# B&R Automation Studio project NAEUL004C00R13L518F00 (part 22)

#### Act_OptP0938FBCtrl1.st
```iecst
ACTION Act_OptP0938FBCtrl1:

	//Motor
	fbJogSlowToFastDlyTm.PT	:= T#2s;
	fbJogSlowToFastDlyTm;
	fbLmtRstTm;

	IF EDGENEG(bMagAWSelfTest) THEN
		eMag1AWEngageAct	:= PneuActIdle;
		eMagAWOpen1Act	:= MagAWActIdle;
	END_IF

	IF bMagAWSelfTest = FALSE THEN

		usiMagAWSelfTestStep := 0;
		//Interruption
		IF tyP0938MagAW.tyMagAW1.tyBtnMtrGearEngage.bRtCompl = TRUE AND (EDGENEG(p_tyDI.bMagPresentSen1) OR EDGEPOS(p_eMag1AWEngageStatus = Error)) THEN
			tyP0938MagAW.tyMotionStd1.tyBtnStop.bRtCompl	:= TRUE;
		END_IF

		IF EDGEPOS((p_udiMagAWOpen1AxisErrID = 21570 OR p_udiMagAWOpen1AxisErrID = 21571) AND tyP0938MagAW.tyMotionStd1.tyBtnJogOpen.bValue = FALSE AND tyP0938MagAW.tyMotionStd1.tyBtnJogClose.bValue = FALSE) THEN
			fbLmtRstTm.IN	:= TRUE;
		END_IF

		IF fbLmtRstTm.Q = TRUE THEN
			tyP0938MagAW.tyMotionStd1.tyBtnRst.bRtCompl		:= TRUE;
		END_IF

		IF (tyP0938MagAW.tyMotionStd1.tyBtnJogOpen.bValue = FALSE AND tyP0938MagAW.tyMotionStd1.tyBtnJogClose.bValue = FALSE) AND (p_bMagAWOpen1Jogging = TRUE) THEN
			bJogStopMagAW1	:= TRUE;
		END_IF

		IF tyP0938MagAW.tyMotionStd1.tyBtnStop.bRtCompl = TRUE THEN

			IF tyP0938MagAW.tyMagAW1.tyBtnMtrGearEngage.bRtCompl = TRUE THEN
				eMagAWOpen1Act		:= MagAWActEngageStop;
				eMag1AWEngageAct	:= PneuActIdle;
			ELSE
				eMagAWOpen1Act		:= MagAWActStop;
			END_IF

			IF (p_eMagAWOpen1Stat = MagAWActStop AND p_eMagAWOpen1Status = Done) OR (p_eMagAWOpen1Stat = MagAWActEngageStop AND p_eMagAWOpen1Status = Done) THEN
				eMagAWOpen1Act	:= MagAWActIdle;

				tyP0938MagAW.tyMotionStd1.tyBtnStop.bRtCompl		:= FALSE;
				tyP0938MagAW.tyMotionStd1.tyBtnJogOpen.bRtCompl		:= FALSE;
				tyP0938MagAW.tyMotionStd1.tyBtnJogClose.bRtCompl	:= FALSE;
				tyP0938MagAW.tyMotionStd1.tyBtnOrigin.bRtCompl		:= FALSE;
				tyP0938MagAW.tyMotionStd1.tyBtnMovAbs.bRtCompl		:= FALSE;
				tyP0938MagAW.tyMotionStd1.tyBtnMovRel.bRtCompl		:= FALSE;
				tyP0938MagAW.tyMagAW1.tyBtnGo.bRtCompl				:= FALSE;
				tyP0938MagAW.tyMagAW1.tyBtnMtrGearEngage.bRtCompl	:= FALSE;

				tyP0938MagAW.tyMotionStd1.tyBtnStop.bValue			:= TRUE;
				tyP0938MagAW.tyMotionStd1.tyBtnJogOpen.bValue		:= FALSE;
				tyP0938MagAW.tyMotionStd1.tyBtnJogClose.bValue		:= FALSE;
				tyP0938MagAW.tyMotionStd1.tyBtnOrigin.bValue		:= FALSE;
				tyP0938MagAW.tyMotionStd1.tyBtnMovAbs.bValue		:= FALSE;
				tyP0938MagAW.tyMotionStd1.tyBtnMovRel.bValue		:= FALSE;
				tyP0938MagAW.tyMagAW1.tyBtnGo.bValue				:= FALSE;
				tyP0938MagAW.tyMagAW1.tyBtnMtrGearEngage.bValue		:= FALSE;

				tyP0938MagAW.tyMotionStd1.tyBtnStop.bRtLk			:= TRUE;
				tyP0938MagAW.tyMotionStd1.tyBtnJogOpen.bRtLk		:= FALSE;
				tyP0938MagAW.tyMotionStd1.tyBtnJogClose.bRtLk		:= FALSE;
				tyP0938MagAW.tyMotionStd1.tyBtnOrigin.bRtLk			:= FALSE;
				tyP0938MagAW.tyMotionStd1.tyBtnMovAbs.bRtLk			:= FALSE;
				tyP0938MagAW.tyMotionStd1.tyBtnMovRel.bRtLk			:= FALSE;
				tyP0938MagAW.tyMagAW1.tyBtnGo.bRtLk					:= FALSE;
				tyP0938MagAW.tyMagAW1.tyBtnMtrGearEngage.bRtLk		:= FALSE;
			END_IF

		ELSIF (tyP0938MagAW.tyMotionStd1.tyBtnJogOpen.bRtCompl = TRUE) OR (tyP0938MagAW.tyMotionStd1.tyBtnJogClose.bRtCompl = TRUE) OR (bJogStopMagAW1 = TRUE) THEN
			bJogSlow					:= FALSE;
			bJogFast					:= FALSE;
			fbJogSlowToFastDlyTm.IN		:= FALSE;

			eMagAWOpen1Act	:= MagAWActJogStop;

			IF p_eMagAWOpen1Stat = MagAWActJogStop AND p_eMagAWOpen1Status = Done THEN
				eMagAWOpen1Act	:= MagAWActIdle;

				bJogStopMagAW1	:= FALSE;

				tyP0938MagAW.tyMotionStd1.tyBtnStop.bRtCompl		:= FALSE;
				tyP0938MagAW.tyMotionStd1.tyBtnJogOpen.bRtCompl		:= FALSE;
				tyP0938MagAW.tyMotionStd1.tyBtnJogClose.bRtCompl	:= FALSE;
				tyP0938MagAW.tyMotionStd1.tyBtnOrigin.bRtCompl		:= FALSE;
				tyP0938MagAW.tyMotionStd1.tyBtnMovAbs.bRtCompl		:= FALSE;
				tyP0938MagAW.tyMotionStd1.tyBtnMovRel.bRtCompl		:= FALSE;
				tyP0938MagAW.tyMagAW1.tyBtnGo.bRtCompl				:= FALSE;

				tyP0938MagAW.tyMotionStd1.tyBtnStop.bValue			:= TRUE;
				tyP0938MagAW.tyMotionStd1.tyBtnJogOpen.bValue		:= FALSE;
				tyP0938MagAW.tyMotionStd1.tyBtnJogClose.bValue		:= FALSE;
				tyP0938MagAW.tyMotionStd1.tyBtnOrigin.bValue		:= FALSE;
				tyP0938MagAW.tyMotionStd1.tyBtnMovAbs.bValue		:= FALSE;
				tyP0938MagAW.tyMotionStd1.tyBtnMovRel.bValue		:= FALSE;
				tyP0938MagAW.tyMagAW1.tyBtnGo.bValue				:= FALSE;

				tyP0938MagAW.tyMotionStd1.tyBtnStop.bRtLk			:= TRUE;
				tyP0938MagAW.tyMotionStd1.tyBtnJogOpen.bRtLk		:= FALSE;
				tyP0938MagAW.tyMotionStd1.tyBtnJogClose.bRtLk		:= FALSE;
				tyP0938MagAW.tyMotionStd1.tyBtnOrigin.bRtLk			:= FALSE;
				tyP0938MagAW.tyMotionStd1.tyBtnMovAbs.bRtLk			:= FALSE;
				tyP0938MagAW.tyMotionStd1.tyBtnMovRel.bRtLk			:= FALSE;
				tyP0938MagAW.tyMagAW1.tyBtnGo.bRtLk					:= FALSE;
			END_IF

		ELSIF tyP0938MagAW.tyMotionStd1.tyBtnPwr.bRtCompl = TRUE THEN
			tyP0938MagAW.tyMotionStd1.tyBtnPwr.bRtLk	:= TRUE;

			IF tyP0938MagAW.tyMotionStd1.tyBtnPwr.bValue = TRUE THEN
				eMagAWOpen1Act	:= MagAWActPwrOn;

				IF p_eMagAWOpen1Stat = MagAWActPwrOn AND p_eMagAWOpen1Status = Done THEN
					eMagAWOpen1Act	:= MagAWActIdle;

					tyP0938MagAW.tyMotionStd1.tyBtnPwr.bRtCompl	:= FALSE;
					tyP0938MagAW.tyMotionStd1.tyBtnPwr.bRtLk	:= FALSE;
				END_IF
			ELSE
				eMagAWOpen1Act	:= MagAWActPwrOff;

				IF p_eMagAWOpen1Stat = MagAWActPwrOff AND p_eMagAWOpen1Status = Done THEN
					eMagAWOpen1Act	:= MagAWActIdle;

					tyP0938MagAW.tyMotionStd1.tyBtnPwr.bRtCompl	:= FALSE;
					tyP0938MagAW.tyMotionStd1.tyBtnPwr.bRtLk	:= FALSE;
				END_IF
			END_IF

		ELSIF tyP0938MagAW.tyMotionStd1.tyBtnOrigin.bRtCompl = TRUE THEN
			tyP0938MagAW.tyMotionStd1.tyBtnOrigin.bValue	:= TRUE;
			tyP0938MagAW.tyMotionStd1.tyBtnStop.bValue		:= FALSE;

			tyP0938MagAW.tyMotionStd1.tyBtnOrigin.bRtLk		:= TRUE;
			tyP0938MagAW.tyMotionStd1.tyBtnStop.bRtLk		:= FALSE;

			eMagAWOpen1Act	:= MagAWActHoming;

			IF p_eMagAWOpen1Stat = MagAWActHoming AND p_eMagAWOpen1Status = Done THEN
				eMagAWOpen1Act	:= MagAWActIdle;

				tyP0938MagAW.tyMotionStd1.tyBtnOrigin.bRtCompl	:= FALSE;
				tyP0938MagAW.tyMotionStd1.tyBtnOrigin.bValue	:= FALSE;
				tyP0938MagAW.tyMotionStd1.tyBtnStop.bValue		:= TRUE;

				tyP0938MagAW.tyMotionStd1.tyBtnOrigin.bRtLk		:= FALSE;
				tyP0938MagAW.tyMotionStd1.tyBtnStop.bRtLk		:= TRUE;
			END_IF

		ELSIF tyP0938MagAW.tyMotionStd1.tyBtnRst.bRtCompl = TRUE THEN
			tyP0938MagAW.tyMotionStd1.tyBtnRst.bValue	:= TRUE;
			tyP0938MagAW.tyMotionStd1.tyBtnRst.bRtLk	:= TRUE;

			eMagAWOpen1Act	:= MagAWActRstAxisErr;

			IF p_eMagAWOpen1Stat = MagAWActRstAxisErr AND p_eMagAWOpen1Status = Done THEN
				eMagAWOpen1Act	:= MagAWActIdle;

				tyP0938MagAW.tyMotionStd1.tyBtnRst.bRtCompl	:= FALSE;
				tyP0938MagAW.tyMotionStd1.tyBtnRst.bValue	:= FALSE;
				tyP0938MagAW.tyMotionStd1.tyBtnRst.bRtLk	:= FALSE;

				fbLmtRstTm.IN	:= FALSE;
			END_IF

		ELSIF tyP0938MagAW.tyMagAW1.tyBtnGo.bRtCompl = TRUE THEN
			tyP0938MagAW.tyMagAW1.tyBtnGo.bValue		:= TRUE;
			tyP0938MagAW.tyMotionStd1.tyBtnStop.bValue	:= FALSE;

			tyP0938MagAW.tyMagAW1.tyBtnGo.bRtLk			:= TRUE;
			tyP0938MagAW.tyMotionStd1.tyBtnStop.bRtLk	:= FALSE;

			diMnlMagAW1GoWidth	:= tyP0938MagAW.tyMagAW1.tyNumNewWidth.diValue;
			diMnlMagAW1NomSpd	:= tyP0938MagAW.tyMotionStd1.tyNumNomSpd.diValue;

			eMagAWOpen1Act	:= MagAWActGoWidth;

			IF p_eMagAWOpen1Stat = MagAWActGoWidth AND p_eMagAWOpen1Status = Done THEN
				eMagAWOpen1Act	:= MagAWActIdle;

				tyP0938MagAW.tyMagAW1.tyBtnGo.bRtCompl		:= FALSE;
				tyP0938MagAW.tyMagAW1.tyBtnGo.bValue		:= FALSE;
				tyP0938MagAW.tyMotionStd1.tyBtnStop.bValue	:= TRUE;

				tyP0938MagAW.tyMagAW1.tyBtnGo.bRtLk			:= FALSE;
				tyP0938MagAW.tyMotionStd1.tyBtnStop.bRtLk	:= TRUE;
			END_IF

		ELSIF tyP0938MagAW.tyMotionStd1.tyBtnMovAbs.bRtCompl = TRUE THEN
			tyP0938MagAW.tyMotionStd1.tyBtnMovAbs.bValue	:= TRUE;
			tyP0938MagAW.tyMotionStd1.tyBtnStop.bValue		:= FALSE;

			tyP0938MagAW.tyMotionStd1.tyBtnMovAbs.bRtLk		:= TRUE;
			tyP0938MagAW.tyMotionStd1.tyBtnStop.bRtLk		:= FALSE;

			diMnlMagAW1TargetPos	:= tyP0938MagAW.tyMotionStd1.tyNumTargetPos.diValue;
			diMnlMagAW1NomSpd		:= tyP0938MagAW.tyMotionStd1.tyNumNomSpd.diValue;

			eMagAWOpen1Act	:= MagAWActMovAbs;

			IF p_eMagAWOpen1Stat = MagAWActMovAbs AND p_eMagAWOpen1Status = Done THEN
				eMagAWOpen1Act	:= MagAWActIdle;

				tyP0938MagAW.tyMotionStd1.tyBtnMovAbs.bRtCompl	:= FALSE;
				tyP0938MagAW.tyMotionStd1.tyBtnMovAbs.bValue	:= FALSE;
				tyP0938MagAW.tyMotionStd1.tyBtnStop.bValue		:= TRUE;

				tyP0938MagAW.tyMotionStd1.tyBtnMovAbs.bRtLk		:= FALSE;
				tyP0938MagAW.tyMotionStd1.tyBtnStop.bRtLk		:= TRUE;
			END_IF

		ELSIF tyP0938MagAW.tyMotionStd1.tyBtnMovRel.bRtCompl = TRUE THEN
			tyP0938MagAW.tyMotionStd1.tyBtnMovRel.bValue	:= TRUE;
			tyP0938MagAW.tyMotionStd1.tyBtnStop.bValue		:= FALSE;

			tyP0938MagAW.tyMotionStd1.tyBtnMovRel.bRtLk		:= TRUE;
			tyP0938MagAW.tyMotionStd1.tyBtnStop.bRtLk		:= FALSE;

			diMnlMagAW1StepSize	:= tyP0938MagAW.tyMotionStd1.tyNumStepSize.diValue;
			diMnlMagAW1NomSpd	:= tyP0938MagAW.tyMotionStd1.tyNumNomSpd.diValue;

			eMagAWOpen1Act	:= MagAWActMovRel;

			IF p_eMagAWOpen1Stat = MagAWActMovRel AND p_eMagAWOpen1Status = Done THEN
				eMagAWOpen1Act	:= MagAWActIdle;

				tyP0938MagAW.tyMotionStd1.tyBtnMovRel.bRtCompl	:= FALSE;
				tyP0938MagAW.tyMotionStd1.tyBtnMovRel.bValue	:= FALSE;
				tyP0938MagAW.tyMotionStd1.tyBtnStop.bValue		:= TRUE;

				tyP0938MagAW.tyMotionStd1.tyBtnMovRel.bRtLk		:= FALSE;
				tyP0938MagAW.tyMotionStd1.tyBtnStop.bRtLk		:= TRUE;
			END_IF

		ELSIF (tyP0938MagAW.tyMotionStd1.tyBtnJogOpen.bValue = TRUE) AND (fbJogSlowToFastDlyTm.Q = FALSE) AND (bJogSlow = FALSE) THEN
			tyP0938MagAW.tyMotionStd1.tyBtnStop.bValue	:= FALSE;
			tyP0938MagAW.tyMotionStd1.tyBtnStop.bRtLk	:= FALSE;

			fbJogSlowToFastDlyTm.IN	:= TRUE;

			diMnlMagAW1JogSpd	:= tyP0938MagAW.tyMotionStd1.tyNumSlwSpd.diValue;

			eMagAWOpen1Act	:= MagAWActJogOpen;

			IF p_eMagAWOpen1Stat = MagAWActJogOpen AND p_eMagAWOpen1Status = Done THEN
				eMagAWOpen1Act				:= MagAWActIdle;
				bJogSlow				:= TRUE;
			ELSIF p_eMagAWOpen1Status = Error THEN
				fbJogSlowToFastDlyTm.IN	:= FALSE;
				bJogSlow				:= TRUE;
			END_IF

		ELSIF (tyP0938MagAW.tyMotionStd1.tyBtnJogOpen.bValue = TRUE) AND (fbJogSlowToFastDlyTm.Q = TRUE) AND (bJogFast = FALSE) THEN
			tyP0938MagAW.tyMotionStd1.tyBtnStop.bValue	:= FALSE;
			tyP0938MagAW.tyMotionStd1.tyBtnStop.bRtLk	:= FALSE;

			fbJogSlowToFastDlyTm.IN	:= TRUE;

			diMnlMagAW1JogSpd	:= tyP0938MagAW.tyMotionStd1.tyNumNomSpd.diValue;

			eMagAWOpen1Act	:= MagAWActJogOpen;

			IF p_eMagAWOpen1Stat = MagAWActJogOpen AND p_eMagAWOpen1Status = Done THEN
				eMagAWOpen1Act				:= MagAWActIdle;
				bJogFast				:= TRUE;
			ELSIF p_eMagAWOpen1Status = Error THEN
				fbJogSlowToFastDlyTm.IN	:= FALSE;
				bJogFast				:= TRUE;
			END_IF

		ELSIF (tyP0938MagAW.tyMotionStd1.tyBtnJogClose.bValue = TRUE) AND (fbJogSlowToFastDlyTm.Q = FALSE) AND (bJogSlow = FALSE) THEN
			tyP0938MagAW.tyMotionStd1.tyBtnStop.bValue	:= FALSE;
			tyP0938MagAW.tyMotionStd1.tyBtnStop.bRtLk	:= FALSE;

			fbJogSlowToFastDlyTm.IN	:= TRUE;

			diMnlMagAW1JogSpd	:= tyP0938MagAW.tyMotionStd1.tyNumSlwSpd.diValue;

			eMagAWOpen1Act	:= MagAWActJogClose;

			IF p_eMagAWOpen1Stat = MagAWActJogClose AND p_eMagAWOpen1Status = Done THEN
				eMagAWOpen1Act				:= MagAWActIdle;
				bJogSlow				:= TRUE;
			ELSIF p_eMagAWOpen1Status = Error THEN
				fbJogSlowToFastDlyTm.IN	:= FALSE;
				bJogSlow				:= TRUE;
			END_IF

		ELSIF (tyP0938MagAW.tyMotionStd1.tyBtnJogClose.bValue = TRUE) AND (fbJogSlowToFastDlyTm.Q = TRUE) AND (bJogFast = FALSE) THEN
			tyP0938MagAW.tyMotionStd1.tyBtnStop.bValue	:= FALSE;
			tyP0938MagAW.tyMotionStd1.tyBtnStop.bRtLk	:= FALSE;

			fbJogSlowToFastDlyTm.IN	:= TRUE;

			diMnlMagAW1JogSpd	:= tyP0938MagAW.tyMotionStd1.tyNumNomSpd.diValue;

			eMagAWOpen1Act	:= MagAWActJogClose;

			IF p_eMagAWOpen1Stat = MagAWActJogClose AND p_eMagAWOpen1Status = Done THEN
				eMagAWOpen1Act				:= MagAWActIdle;
				bJogFast				:= TRUE;
			ELSIF p_eMagAWOpen1Status = Error THEN
				fbJogSlowToFastDlyTm.IN	:= FALSE;
				bJogFast				:= TRUE;
			END_IF

		ELSIF tyP0938MagAW.tyMagAW1.tyBtnMtrGearEngage.bRtCompl = TRUE THEN
			tyP0938MagAW.tyMagAW1.tyBtnMtrGearEngage.bValue	:= TRUE;
			tyP0938MagAW.tyMotionStd1.tyBtnStop.bValue		:= FALSE;

			tyP0938MagAW.tyMagAW1.tyBtnMtrGearEngage.bRtLk	:= TRUE;
			tyP0938MagAW.tyMotionStd1.tyBtnStop.bRtLk		:= FALSE;

			eMagAWOpen1Act	:= MagAWActEngage;

			IF p_bMagAWOpen1Engaging = TRUE THEN
				eMag1AWEngageAct	:= PneuActExt;

				tyP0938MagAW.tyMagAW1.tyBtnEngage.bValue	:= TRUE;
				tyP0938MagAW.tyMagAW1.tyBtnDisengage.bValue	:= FALSE;
			END_IF

			IF (p_eMagAWOpen1Stat = MagAWActEngage AND p_eMagAWOpen1Status = Done) AND (p_eMag1AWEngageStat = PneuActExt AND p_eMag1AWEngageStatus = Done) THEN
				eMagAWOpen1Act		:= MagAWActIdle;
				eMag1AWEngageAct	:= PneuActIdle;

				tyP0938MagAW.tyMagAW1.tyBtnMtrGearEngage.bRtCompl	:= FALSE;
				tyP0938MagAW.tyMagAW1.tyBtnMtrGearEngage.bValue		:= FALSE;
				tyP0938MagAW.tyMotionStd1.tyBtnStop.bValue			:= TRUE;

				tyP0938MagAW.tyMagAW1.tyBtnMtrGearEngage.bRtLk		:= FALSE;
				tyP0938MagAW.tyMotionStd1.tyBtnStop.bRtLk			:= TRUE;
			END_IF

		END_IF

		//Pneumatic
		IF p_bMag1AWEngageTwoCtrlOut = FALSE THEN

			IF tyP0938MagAW.tyMagAW1.tyBtnDisengage.bRtCompl = TRUE THEN
				tyP0938MagAW.tyMagAW1.tyBtnDisengage.bValue	:= TRUE;
				tyP0938MagAW.tyMagAW1.tyBtnEngage.bValue	:= FALSE;

				eMag1AWEngageAct	:= PneuActSetRet;

				IF p_eMag1AWEngageStat = PneuActSetRet AND p_eMag1AWEngageStatus = Done THEN
					eMag1AWEngageAct	:= PneuActIdle;

					tyP0938MagAW.tyMagAW1.tyBtnDisengage.bRtCompl	:= FALSE;
				END_IF

			ELSIF tyP0938MagAW.tyMagAW1.tyBtnEngage.bRtCompl = TRUE THEN
				tyP0938MagAW.tyMagAW1.tyBtnEngage.bValue	:= TRUE;
				tyP0938MagAW.tyMagAW1.tyBtnDisengage.bValue	:= FALSE;

				eMag1AWEngageAct	:= PneuActSetExt;

				IF p_eMag1AWEngageStat = PneuActSetExt AND p_eMag1AWEngageStatus = Done THEN
					eMag1AWEngageAct	:= PneuActIdle;

					tyP0938MagAW.tyMagAW1.tyBtnEngage.bRtCompl	:= FALSE;
				END_IF

			END_IF

		ELSE

			IF (tyP0938MagAW.tyMagAW1.tyBtnDisengage.bRtCompl = TRUE) OR (tyP0938MagAW.tyMagAW1.tyBtnEngage.bRtCompl = TRUE) THEN

				IF (tyP0938MagAW.tyMagAW1.tyBtnDisengage.bValue = TRUE) AND (tyP0938MagAW.tyMagAW1.tyBtnEngage.bValue = TRUE) THEN
					eMag1AWEngageAct	:= PneuActSetAll;

					IF p_eMag1AWEngageStat = PneuActSetAll AND p_eMag1AWEngageStatus = Done THEN
						eMag1AWEngageAct	:= PneuActIdle;

						tyP0938MagAW.tyMagAW1.tyBtnDisengage.bRtCompl	:= FALSE;
						tyP0938MagAW.tyMagAW1.tyBtnEngage.bRtCompl		:= FALSE;
					END_IF

				ELSIF (tyP0938MagAW.tyMagAW1.tyBtnDisengage.bValue = TRUE) AND (tyP0938MagAW.tyMagAW1.tyBtnEngage.bValue = FALSE) THEN
					eMag1AWEngageAct	:= PneuActSetRet;

					IF p_eMag1AWEngageStat = PneuActSetRet AND p_eMag1AWEngageStatus = Done THEN
						eMag1AWEngageAct	:= PneuActIdle;

						tyP0938MagAW.tyMagAW1.tyBtnDisengage.bRtCompl	:= FALSE;
						tyP0938MagAW.tyMagAW1.tyBtnEngage.bRtCompl		:= FALSE;
					END_IF

				ELSIF (tyP0938MagAW.tyMagAW1.tyBtnDisengage.bValue = FALSE) AND (tyP0938MagAW.tyMagAW1.tyBtnEngage.bValue = TRUE) THEN
					eMag1AWEngageAct	:= PneuActSetExt;

					IF p_eMag1AWEngageStat = PneuActSetExt AND p_eMag1AWEngageStatus = Done THEN
						eMag1AWEngageAct	:= PneuActIdle;

						tyP0938MagAW.tyMagAW1.tyBtnDisengage.bRtCompl	:= FALSE;
						tyP0938MagAW.tyMagAW1.tyBtnEngage.bRtCompl		:= FALSE;
					END_IF

				ELSE
					eMag1AWEngageAct	:= PneuActRstAll;

					IF p_eMag1AWEngageStat = PneuActRstAll AND p_eMag1AWEngageStatus = Done THEN
						eMag1AWEngageAct	:= PneuActIdle;

						tyP0938MagAW.tyMagAW1.tyBtnDisengage.bRtCompl	:= FALSE;
						tyP0938MagAW.tyMagAW1.tyBtnEngage.bRtCompl		:= FALSE;
					END_IF

				END_IF

			END_IF

		END_IF

	ELSE

		CASE usiMagAWSelfTestStep OF

			0: IF p_bMagConv2Clp1ClprFixClampCtrl THEN

					eMagAWOpen1Act	:= MagAWActEngage;

						eMag1AWEngageAct	:= PneuActExt;

						IF (p_eMagAWOpen1Stat = MagAWActEngage AND p_eMagAWOpen1Status = Done)
							AND (p_eMag1AWEngageStat = PneuActExt AND p_eMag1AWEngageStatus = Done)
						THEN
							eMagAWOpen1Act		:= MagAWActIdle;
							eMag1AWEngageAct	:= PneuActIdle;
							usiMagAWSelfTestStep := 10;
						END_IF

				END_IF

			10:
				eMagAWOpen1Act	:= MagAWActHoming;

				IF p_eMagAWOpen1Stat = MagAWActHoming AND p_eMagAWOpen1Status = Done THEN
					eMagAWOpen1Act	:= MagAWActIdle;
					usiMagAWSelfTestStep := 20;
				END_IF

			20:

				diMnlMagAW1GoWidth	:= tyP0938MagAW.tyMagAW1.tyNumNewWidth.diValue;
				diMnlMagAW1NomSpd		:= tyP0938MagAW.tyMotionStd1.tyNumNomSpd.diValue;
				eMagAWOpen1Act	:= MagAWActGoWidth;

				IF p_eMagAWOpen1Stat = MagAWActGoWidth AND p_eMagAWOpen1Status = Done THEN
					eMagAWOpen1Act	:= MagAWActIdle;
					usiMagAWSelfTestStep := 30;
				END_IF

			30:
				eMag1AWEngageAct	:= PneuActSetRet;

				IF p_eMag1AWEngageStat = PneuActSetRet AND p_eMag1AWEngageStatus = Done THEN
					eMag1AWEngageAct	:= PneuActIdle;
					usiMagAWSelfTestStep := 40;
				END_IF

			40:
				fbMagAWSelfTestTim(IN:= TRUE);
				IF fbMagAWSelfTestTim.Q THEN
						usiMagAWSelfTestStep := 0;
						fbMagAWSelfTestTim(IN:= FALSE);
					END_IF
		END_CASE
	END_IF

END_ACTION
```

#### Act_OptP0938FBCtrl2.st
```iecst
ACTION Act_OptP0938FBCtrl2:

	//Motor
	fbJogSlowToFastDlyTm.PT	:= T#2s;
	fbJogSlowToFastDlyTm;
	fbLmtRstTm;

	IF EDGENEG(bMagAWSelfTest) THEN
		eMag2AWEngageAct	:= PneuActIdle;
		eMagAWOpen2Act	:= MagAWActIdle;
	END_IF

	IF bMagAWSelfTest = FALSE THEN
		usiMagAWSelfTestStep1 := 0;
		//Interruption
		IF tyP0938MagAW.tyMagAW2.tyBtnMtrGearEngage.bRtCompl = TRUE AND (EDGENEG(p_tyDI.bMagPresentSen2) OR EDGEPOS(p_eMag2AWEngageStatus = Error)) THEN
			tyP0938MagAW.tyMotionStd2.tyBtnStop.bRtCompl	:= TRUE;
		END_IF

		IF EDGEPOS((p_udiMagAWOpen2AxisErrID = 21570 OR p_udiMagAWOpen2AxisErrID = 21571) AND tyP0938MagAW.tyMotionStd2.tyBtnJogOpen.bValue = FALSE AND tyP0938MagAW.tyMotionStd2.tyBtnJogClose.bValue = FALSE) THEN
			fbLmtRstTm.IN	:= TRUE;
		END_IF

		IF fbLmtRstTm.Q = TRUE THEN
			tyP0938MagAW.tyMotionStd2.tyBtnRst.bRtCompl		:= TRUE;
		END_IF

		IF (tyP0938MagAW.tyMotionStd2.tyBtnJogOpen.bValue = FALSE AND tyP0938MagAW.tyMotionStd2.tyBtnJogClose.bValue = FALSE) AND (p_bMagAWOpen2Jogging = TRUE) THEN
			bJogStopMagAW2	:= TRUE;
		END_IF

		IF tyP0938MagAW.tyMotionStd2.tyBtnStop.bRtCompl = TRUE THEN

			IF tyP0938MagAW.tyMagAW2.tyBtnMtrGearEngage.bRtCompl = TRUE THEN
				eMagAWOpen2Act		:= MagAWActEngageStop;
				eMag2AWEngageAct	:= PneuActIdle;
			ELSE
				eMagAWOpen2Act		:= MagAWActStop;
			END_IF

			IF (p_eMagAWOpen2Stat = MagAWActStop AND p_eMagAWOpen2Status = Done) OR (p_eMagAWOpen2Stat = MagAWActEngageStop AND p_eMagAWOpen2Status = Done) THEN
				eMagAWOpen2Act	:= MagAWActIdle;

				tyP0938MagAW.tyMotionStd2.tyBtnStop.bRtCompl		:= FALSE;
				tyP0938MagAW.tyMotionStd2.tyBtnJogOpen.bRtCompl		:= FALSE;
				tyP0938MagAW.tyMotionStd2.tyBtnJogClose.bRtCompl	:= FALSE;
				tyP0938MagAW.tyMotionStd2.tyBtnOrigin.bRtCompl		:= FALSE;
				tyP0938MagAW.tyMotionStd2.tyBtnMovAbs.bRtCompl		:= FALSE;
				tyP0938MagAW.tyMotionStd2.tyBtnMovRel.bRtCompl		:= FALSE;
				tyP0938MagAW.tyMagAW2.tyBtnGo.bRtCompl				:= FALSE;
				tyP0938MagAW.tyMagAW2.tyBtnMtrGearEngage.bRtCompl	:= FALSE;

				tyP0938MagAW.tyMotionStd2.tyBtnStop.bValue			:= TRUE;
				tyP0938MagAW.tyMotionStd2.tyBtnJogOpen.bValue		:= FALSE;
				tyP0938MagAW.tyMotionStd2.tyBtnJogClose.bValue		:= FALSE;
				tyP0938MagAW.tyMotionStd2.tyBtnOrigin.bValue		:= FALSE;
				tyP0938MagAW.tyMotionStd2.tyBtnMovAbs.bValue		:= FALSE;
				tyP0938MagAW.tyMotionStd2.tyBtnMovRel.bValue		:= FALSE;
				tyP0938MagAW.tyMagAW2.tyBtnGo.bValue				:= FALSE;
				tyP0938MagAW.tyMagAW2.tyBtnMtrGearEngage.bValue		:= FALSE;

				tyP0938MagAW.tyMotionStd2.tyBtnStop.bRtLk			:= TRUE;
				tyP0938MagAW.tyMotionStd2.tyBtnJogOpen.bRtLk		:= FALSE;
				tyP0938MagAW.tyMotionStd2.tyBtnJogClose.bRtLk		:= FALSE;
				tyP0938MagAW.tyMotionStd2.tyBtnOrigin.bRtLk			:= FALSE;
				tyP0938MagAW.tyMotionStd2.tyBtnMovAbs.bRtLk			:= FALSE;
				tyP0938MagAW.tyMotionStd2.tyBtnMovRel.bRtLk			:= FALSE;
				tyP0938MagAW.tyMagAW2.tyBtnGo.bRtLk					:= FALSE;
				tyP0938MagAW.tyMagAW2.tyBtnMtrGearEngage.bRtLk		:= FALSE;
			END_IF

		ELSIF (tyP0938MagAW.tyMotionStd2.tyBtnJogOpen.bRtCompl = TRUE) OR (tyP0938MagAW.tyMotionStd2.tyBtnJogClose.bRtCompl = TRUE) OR (bJogStopMagAW2 = TRUE) THEN
			bJogSlow					:= FALSE;
			bJogFast					:= FALSE;
			fbJogSlowToFastDlyTm.IN		:= FALSE;

			eMagAWOpen2Act	:= MagAWActJogStop;

			IF p_eMagAWOpen2Stat = MagAWActJogStop AND p_eMagAWOpen2Status = Done THEN
				eMagAWOpen2Act	:= MagAWActIdle;

				bJogStopMagAW2	:= FALSE;

				tyP0938MagAW.tyMotionStd2.tyBtnStop.bRtCompl		:= FALSE;
				tyP0938MagAW.tyMotionStd2.tyBtnJogOpen.bRtCompl		:= FALSE;
				tyP0938MagAW.tyMotionStd2.tyBtnJogClose.bRtCompl	:= FALSE;
				tyP0938MagAW.tyMotionStd2.tyBtnOrigin.bRtCompl		:= FALSE;
				tyP0938MagAW.tyMotionStd2.tyBtnMovAbs.bRtCompl		:= FALSE;
				tyP0938MagAW.tyMotionStd2.tyBtnMovRel.bRtCompl		:= FALSE;
				tyP0938MagAW.tyMagAW2.tyBtnGo.bRtCompl				:= FALSE;

				tyP0938MagAW.tyMotionStd2.tyBtnStop.bValue			:= TRUE;
				tyP0938MagAW.tyMotionStd2.tyBtnJogOpen.bValue		:= FALSE;
				tyP0938MagAW.tyMotionStd2.tyBtnJogClose.bValue		:= FALSE;
				tyP0938MagAW.tyMotionStd2.tyBtnOrigin.bValue		:= FALSE;
				tyP0938MagAW.tyMotionStd2.tyBtnMovAbs.bValue		:= FALSE;
				tyP0938MagAW.tyMotionStd2.tyBtnMovRel.bValue		:= FALSE;
				tyP0938MagAW.tyMagAW2.tyBtnGo.bValue				:= FALSE;

				tyP0938MagAW.tyMotionStd2.tyBtnStop.bRtLk			:= TRUE;
				tyP0938MagAW.tyMotionStd2.tyBtnJogOpen.bRtLk		:= FALSE;
				tyP0938MagAW.tyMotionStd2.tyBtnJogClose.bRtLk		:= FALSE;
				tyP0938MagAW.tyMotionStd2.tyBtnOrigin.bRtLk			:= FALSE;
				tyP0938MagAW.tyMotionStd2.tyBtnMovAbs.bRtLk			:= FALSE;
				tyP0938MagAW.tyMotionStd2.tyBtnMovRel.bRtLk			:= FALSE;
				tyP0938MagAW.tyMagAW2.tyBtnGo.bRtLk					:= FALSE;
			END_IF

		ELSIF tyP0938MagAW.tyMotionStd2.tyBtnPwr.bRtCompl = TRUE THEN
			tyP0938MagAW.tyMotionStd2.tyBtnPwr.bRtLk	:= TRUE;

			IF tyP0938MagAW.tyMotionStd2.tyBtnPwr.bValue = TRUE THEN
				eMagAWOpen2Act	:= MagAWActPwrOn;

				IF p_eMagAWOpen2Stat = MagAWActPwrOn AND p_eMagAWOpen2Status = Done THEN
					eMagAWOpen2Act	:= MagAWActIdle;

					tyP0938MagAW.tyMotionStd2.tyBtnPwr.bRtCompl	:= FALSE;
					tyP0938MagAW.tyMotionStd2.tyBtnPwr.bRtLk	:= FALSE;
				END_IF
			ELSE
				eMagAWOpen2Act	:= MagAWActPwrOff;

				IF p_eMagAWOpen2Stat = MagAWActPwrOff AND p_eMagAWOpen2Status = Done THEN
					eMagAWOpen2Act	:= MagAWActIdle;

					tyP0938MagAW.tyMotionStd2.tyBtnPwr.bRtCompl	:= FALSE;
					tyP0938MagAW.tyMotionStd2.tyBtnPwr.bRtLk	:= FALSE;
				END_IF
			END_IF

		ELSIF tyP0938MagAW.tyMotionStd2.tyBtnOrigin.bRtCompl = TRUE THEN
			tyP0938MagAW.tyMotionStd2.tyBtnOrigin.bValue	:= TRUE;
			tyP0938MagAW.tyMotionStd2.tyBtnStop.bValue		:= FALSE;

			tyP0938MagAW.tyMotionStd2.tyBtnOrigin.bRtLk		:= TRUE;
			tyP0938MagAW.tyMotionStd2.tyBtnStop.bRtLk		:= FALSE;

			eMagAWOpen2Act	:= MagAWActHoming;

			IF p_eMagAWOpen2Stat = MagAWActHoming AND p_eMagAWOpen2Status = Done THEN
				eMagAWOpen2Act	:= MagAWActIdle;

				tyP0938MagAW.tyMotionStd2.tyBtnOrigin.bRtCompl	:= FALSE;
				tyP0938MagAW.tyMotionStd2.tyBtnOrigin.bValue	:= FALSE;
				tyP0938MagAW.tyMotionStd2.tyBtnStop.bValue		:= TRUE;

				tyP0938MagAW.tyMotionStd2.tyBtnOrigin.bRtLk		:= FALSE;
				tyP0938MagAW.tyMotionStd2.tyBtnStop.bRtLk		:= TRUE;
			END_IF

		ELSIF tyP0938MagAW.tyMotionStd2.tyBtnRst.bRtCompl = TRUE THEN
			tyP0938MagAW.tyMotionStd2.tyBtnRst.bValue	:= TRUE;
			tyP0938MagAW.tyMotionStd2.tyBtnRst.bRtLk	:= TRUE;

			eMagAWOpen2Act	:= MagAWActRstAxisErr;

			IF p_eMagAWOpen2Stat = MagAWActRstAxisErr AND p_eMagAWOpen2Status = Done THEN
				eMagAWOpen2Act	:= MagAWActIdle;

				tyP0938MagAW.tyMotionStd2.tyBtnRst.bRtCompl	:= FALSE;
				tyP0938MagAW.tyMotionStd2.tyBtnRst.bValue	:= FALSE;
				tyP0938MagAW.tyMotionStd2.tyBtnRst.bRtLk	:= FALSE;

				fbLmtRstTm.IN	:= FALSE;
			END_IF

		ELSIF tyP0938MagAW.tyMagAW2.tyBtnGo.bRtCompl = TRUE THEN
			tyP0938MagAW.tyMagAW2.tyBtnGo.bValue		:= TRUE;
			tyP0938MagAW.tyMotionStd2.tyBtnStop.bValue	:= FALSE;

			tyP0938MagAW.tyMagAW2.tyBtnGo.bRtLk			:= TRUE;
			tyP0938MagAW.tyMotionStd2.tyBtnStop.bRtLk	:= FALSE;

			diMnlMagAW2GoWidth	:= tyP0938MagAW.tyMagAW2.tyNumNewWidth.diValue;
			diMnlMagAW2NomSpd	:= tyP0938MagAW.tyMotionStd2.tyNumNomSpd.diValue;

			eMagAWOpen2Act	:= MagAWActGoWidth;

			IF p_eMagAWOpen2Stat = MagAWActGoWidth AND p_eMagAWOpen2Status = Done THEN
				eMagAWOpen2Act	:= MagAWActIdle;

				tyP0938MagAW.tyMagAW2.tyBtnGo.bRtCompl		:= FALSE;
				tyP0938MagAW.tyMagAW2.tyBtnGo.bValue		:= FALSE;
				tyP0938MagAW.tyMotionStd2.tyBtnStop.bValue	:= TRUE;

				tyP0938MagAW.tyMagAW2.tyBtnGo.bRtLk			:= FALSE;
				tyP0938MagAW.tyMotionStd2.tyBtnStop.bRtLk	:= TRUE;
			END_IF

		ELSIF tyP0938MagAW.tyMotionStd2.tyBtnMovAbs.bRtCompl = TRUE THEN
			tyP0938MagAW.tyMotionStd2.tyBtnMovAbs.bValue	:= TRUE;
			tyP0938MagAW.tyMotionStd2.tyBtnStop.bValue		:= FALSE;

			tyP0938MagAW.tyMotionStd2.tyBtnMovAbs.bRtLk		:= TRUE;
			tyP0938MagAW.tyMotionStd2.tyBtnStop.bRtLk		:= FALSE;

			diMnlMagAW2TargetPos	:= tyP0938MagAW.tyMotionStd2.tyNumTargetPos.diValue;
			diMnlMagAW2NomSpd		:= tyP0938MagAW.tyMotionStd2.tyNumNomSpd.diValue;

			eMagAWOpen2Act	:= MagAWActMovAbs;

			IF p_eMagAWOpen2Stat = MagAWActMovAbs AND p_eMagAWOpen2Status = Done THEN
				eMagAWOpen2Act	:= MagAWActIdle;

				tyP0938MagAW.tyMotionStd2.tyBtnMovAbs.bRtCompl	:= FALSE;
				tyP0938MagAW.tyMotionStd2.tyBtnMovAbs.bValue	:= FALSE;
				tyP0938MagAW.tyMotionStd2.tyBtnStop.bValue		:= TRUE;

				tyP0938MagAW.tyMotionStd2.tyBtnMovAbs.bRtLk		:= FALSE;
				tyP0938MagAW.tyMotionStd2.tyBtnStop.bRtLk		:= TRUE;
			END_IF

		ELSIF tyP0938MagAW.tyMotionStd2.tyBtnMovRel.bRtCompl = TRUE THEN
			tyP0938MagAW.tyMotionStd2.tyBtnMovRel.bValue	:= TRUE;
			tyP0938MagAW.tyMotionStd2.tyBtnStop.bValue		:= FALSE;

			tyP0938MagAW.tyMotionStd2.tyBtnMovRel.bRtLk		:= TRUE;
			tyP0938MagAW.tyMotionStd2.tyBtnStop.bRtLk		:= FALSE;

			diMnlMagAW2StepSize	:= tyP0938MagAW.tyMotionStd2.tyNumStepSize.diValue;
			diMnlMagAW2NomSpd	:= tyP0938MagAW.tyMotionStd2.tyNumNomSpd.diValue;

			eMagAWOpen2Act	:= MagAWActMovRel;

			IF p_eMagAWOpen2Stat = MagAWActMovRel AND p_eMagAWOpen2Status = Done THEN
				eMagAWOpen2Act	:= MagAWActIdle;

				tyP0938MagAW.tyMotionStd2.tyBtnMovRel.bRtCompl	:= FALSE;
				tyP0938MagAW.tyMotionStd2.tyBtnMovRel.bValue	:= FALSE;
				tyP0938MagAW.tyMotionStd2.tyBtnStop.bValue		:= TRUE;

				tyP0938MagAW.tyMotionStd2.tyBtnMovRel.bRtLk		:= FALSE;
				tyP0938MagAW.tyMotionStd2.tyBtnStop.bRtLk		:= TRUE;
			END_IF

		ELSIF (tyP0938MagAW.tyMotionStd2.tyBtnJogOpen.bValue = TRUE) AND (fbJogSlowToFastDlyTm.Q = FALSE) AND (bJogSlow = FALSE) THEN
			tyP0938MagAW.tyMotionStd2.tyBtnStop.bValue	:= FALSE;
			tyP0938MagAW.tyMotionStd2.tyBtnStop.bRtLk	:= FALSE;

			fbJogSlowToFastDlyTm.IN	:= TRUE;

			diMnlMagAW2JogSpd	:= tyP0938MagAW.tyMotionStd2.tyNumSlwSpd.diValue;

			eMagAWOpen2Act	:= MagAWActJogOpen;

			IF p_eMagAWOpen2Stat = MagAWActJogOpen AND p_eMagAWOpen2Status = Done THEN
				eMagAWOpen2Act				:= MagAWActIdle;
				bJogSlow				:= TRUE;
			ELSIF p_eMagAWOpen2Status = Error THEN
				fbJogSlowToFastDlyTm.IN	:= FALSE;
				bJogSlow				:= TRUE;
			END_IF

		ELSIF (tyP0938MagAW.tyMotionStd2.tyBtnJogOpen.bValue = TRUE) AND (fbJogSlowToFastDlyTm.Q = TRUE) AND (bJogFast = FALSE) THEN
			tyP0938MagAW.tyMotionStd2.tyBtnStop.bValue	:= FALSE;
			tyP0938MagAW.tyMotionStd2.tyBtnStop.bRtLk	:= FALSE;

			fbJogSlowToFastDlyTm.IN	:= TRUE;

			diMnlMagAW2JogSpd	:= tyP0938MagAW.tyMotionStd2.tyNumNomSpd.diValue;

			eMagAWOpen2Act	:= MagAWActJogOpen;

			IF p_eMagAWOpen2Stat = MagAWActJogOpen AND p_eMagAWOpen2Status = Done THEN
				eMagAWOpen2Act				:= MagAWActIdle;
				bJogFast				:= TRUE;
			ELSIF p_eMagAWOpen2Status = Error THEN
				fbJogSlowToFastDlyTm.IN	:= FALSE;
				bJogFast				:= TRUE;
			END_IF

		ELSIF (tyP0938MagAW.tyMotionStd2.tyBtnJogClose.bValue = TRUE) AND (fbJogSlowToFastDlyTm.Q = FALSE) AND (bJogSlow = FALSE) THEN
			tyP0938MagAW.tyMotionStd2.tyBtnStop.bValue	:= FALSE;
			tyP0938MagAW.tyMotionStd2.tyBtnStop.bRtLk	:= FALSE;

			fbJogSlowToFastDlyTm.IN	:= TRUE;

			diMnlMagAW2JogSpd	:= tyP0938MagAW.tyMotionStd2.tyNumSlwSpd.diValue;

			eMagAWOpen2Act	:= MagAWActJogClose;

			IF p_eMagAWOpen2Stat = MagAWActJogClose AND p_eMagAWOpen2Status = Done THEN
				eMagAWOpen2Act				:= MagAWActIdle;
				bJogSlow				:= TRUE;
			ELSIF p_eMagAWOpen2Status = Error THEN
				fbJogSlowToFastDlyTm.IN	:= FALSE;
				bJogSlow				:= TRUE;
			END_IF

		ELSIF (tyP0938MagAW.tyMotionStd2.tyBtnJogClose.bValue = TRUE) AND (fbJogSlowToFastDlyTm.Q = TRUE) AND (bJogFast = FALSE) THEN
			tyP0938MagAW.tyMotionStd2.tyBtnStop.bValue	:= FALSE;
			tyP0938MagAW.tyMotionStd2.tyBtnStop.bRtLk	:= FALSE;

			fbJogSlowToFastDlyTm.IN	:= TRUE;

			diMnlMagAW2JogSpd	:= tyP0938MagAW.tyMotionStd2.tyNumNomSpd.diValue;

			eMagAWOpen2Act	:= MagAWActJogClose;

			IF p_eMagAWOpen2Stat = MagAWActJogClose AND p_eMagAWOpen2Status = Done THEN
				eMagAWOpen2Act				:= MagAWActIdle;
				bJogFast				:= TRUE;
			ELSIF p_eMagAWOpen2Status = Error THEN
				fbJogSlowToFastDlyTm.IN	:= FALSE;
				bJogFast				:= TRUE;
			END_IF

		ELSIF tyP0938MagAW.tyMagAW2.tyBtnMtrGearEngage.bRtCompl = TRUE THEN
			tyP0938MagAW.tyMagAW2.tyBtnMtrGearEngage.bValue	:= TRUE;
			tyP0938MagAW.tyMotionStd2.tyBtnStop.bValue		:= FALSE;

			tyP0938MagAW.tyMagAW2.tyBtnMtrGearEngage.bRtLk	:= TRUE;
			tyP0938MagAW.tyMotionStd2.tyBtnStop.bRtLk		:= FALSE;

			eMagAWOpen2Act	:= MagAWActEngage;

			IF p_bMagAWOpen2Engaging = TRUE THEN
				eMag2AWEngageAct	:= PneuActExt;

				tyP0938MagAW.tyMagAW2.tyBtnEngage.bValue	:= TRUE;
				tyP0938MagAW.tyMagAW2.tyBtnDisengage.bValue	:= FALSE;
			END_IF

			IF (p_eMagAWOpen2Stat = MagAWActEngage AND p_eMagAWOpen2Status = Done) AND (p_eMag2AWEngageStat = PneuActExt AND p_eMag2AWEngageStatus = Done) THEN
				eMagAWOpen2Act		:= MagAWActIdle;
				eMag2AWEngageAct	:= PneuActIdle;

				tyP0938MagAW.tyMagAW2.tyBtnMtrGearEngage.bRtCompl	:= FALSE;
				tyP0938MagAW.tyMagAW2.tyBtnMtrGearEngage.bValue		:= FALSE;
				tyP0938MagAW.tyMotionStd2.tyBtnStop.bValue			:= TRUE;

				tyP0938MagAW.tyMagAW2.tyBtnMtrGearEngage.bRtLk		:= FALSE;
				tyP0938MagAW.tyMotionStd2.tyBtnStop.bRtLk			:= TRUE;
			END_IF

		END_IF

		//Pneumatic
		IF p_bMag2AWEngageTwoCtrlOut = FALSE THEN

			IF tyP0938MagAW.tyMagAW2.tyBtnDisengage.bRtCompl = TRUE THEN
				tyP0938MagAW.tyMagAW2.tyBtnDisengage.bValue	:= TRUE;
				tyP0938MagAW.tyMagAW2.tyBtnEngage.bValue	:= FALSE;

				eMag2AWEngageAct	:= PneuActSetRet;

				IF p_eMag2AWEngageStat = PneuActSetRet AND p_eMag2AWEngageStatus = Done THEN
					eMag2AWEngageAct	:= PneuActIdle;

					tyP0938MagAW.tyMagAW2.tyBtnDisengage.bRtCompl	:= FALSE;
				END_IF

			ELSIF tyP0938MagAW.tyMagAW2.tyBtnEngage.bRtCompl = TRUE THEN
				tyP0938MagAW.tyMagAW2.tyBtnEngage.bValue	:= TRUE;
				tyP0938MagAW.tyMagAW2.tyBtnDisengage.bValue	:= FALSE;

				eMag2AWEngageAct	:= PneuActSetExt;

				IF p_eMag2AWEngageStat = PneuActSetExt AND p_eMag2AWEngageStatus = Done THEN
					eMag2AWEngageAct	:= PneuActIdle;

					tyP0938MagAW.tyMagAW2.tyBtnEngage.bRtCompl	:= FALSE;
				END_IF

			END_IF

		ELSE

			IF (tyP0938MagAW.tyMagAW2.tyBtnDisengage.bRtCompl = TRUE) OR (tyP0938MagAW.tyMagAW2.tyBtnEngage.bRtCompl = TRUE) THEN

				IF (tyP0938MagAW.tyMagAW2.tyBtnDisengage.bValue = TRUE) AND (tyP0938MagAW.tyMagAW2.tyBtnEngage.bValue = TRUE) THEN
					eMag2AWEngageAct	:= PneuActSetAll;

					IF p_eMag2AWEngageStat = PneuActSetAll AND p_eMag2AWEngageStatus = Done THEN
						eMag2AWEngageAct	:= PneuActIdle;

						tyP0938MagAW.tyMagAW2.tyBtnDisengage.bRtCompl	:= FALSE;
						tyP0938MagAW.tyMagAW2.tyBtnEngage.bRtCompl		:= FALSE;
					END_IF

				ELSIF (tyP0938MagAW.tyMagAW2.tyBtnDisengage.bValue = TRUE) AND (tyP0938MagAW.tyMagAW2.tyBtnEngage.bValue = FALSE) THEN
					eMag2AWEngageAct	:= PneuActSetRet;

					IF p_eMag2AWEngageStat = PneuActSetRet AND p_eMag2AWEngageStatus = Done THEN
						eMag2AWEngageAct	:= PneuActIdle;

						tyP0938MagAW.tyMagAW2.tyBtnDisengage.bRtCompl	:= FALSE;
						tyP0938MagAW.tyMagAW2.tyBtnEngage.bRtCompl		:= FALSE;
					END_IF

				ELSIF (tyP0938MagAW.tyMagAW2.tyBtnDisengage.bValue = FALSE) AND (tyP0938MagAW.tyMagAW2.tyBtnEngage.bValue = TRUE) THEN
					eMag2AWEngageAct	:= PneuActSetExt;

					IF p_eMag2AWEngageStat = PneuActSetExt AND p_eMag2AWEngageStatus = Done THEN
						eMag2AWEngageAct	:= PneuActIdle;

						tyP0938MagAW.tyMagAW2.tyBtnDisengage.bRtCompl	:= FALSE;
						tyP0938MagAW.tyMagAW2.tyBtnEngage.bRtCompl		:= FALSE;
					END_IF

				ELSE
					eMag2AWEngageAct	:= PneuActRstAll;

					IF p_eMag2AWEngageStat = PneuActRstAll AND p_eMag2AWEngageStatus = Done THEN
						eMag2AWEngageAct	:= PneuActIdle;

						tyP0938MagAW.tyMagAW2.tyBtnDisengage.bRtCompl	:= FALSE;
						tyP0938MagAW.tyMagAW2.tyBtnEngage.bRtCompl		:= FALSE;
					END_IF

				END_IF

			END_IF

		END_IF

	ELSE
		CASE usiMagAWSelfTestStep1 OF

			0: IF p_bMagConv2Clp2ClprFixClampCtrl THEN

					eMagAWOpen2Act	:= MagAWActEngage;

					eMag2AWEngageAct	:= PneuActExt;

					IF (p_eMagAWOpen2Stat = MagAWActEngage AND p_eMagAWOpen2Status = Done)
						AND (p_eMag2AWEngageStat = PneuActExt AND p_eMag2AWEngageStatus = Done)
						THEN
						eMagAWOpen2Act		:= MagAWActIdle;
						eMag2AWEngageAct	:= PneuActIdle;
						usiMagAWSelfTestStep1 := 10;
					END_IF

				END_IF

			10:
				eMagAWOpen2Act	:= MagAWActHoming;

				IF p_eMagAWOpen2Stat = MagAWActHoming AND p_eMagAWOpen2Status = Done THEN
					eMagAWOpen2Act	:= MagAWActIdle;
					usiMagAWSelfTestStep1 := 20;
				END_IF

			20:

				diMnlMagAW2GoWidth	:= tyP0938MagAW.tyMagAW1.tyNumNewWidth.diValue;
				diMnlMagAW2NomSpd		:= tyP0938MagAW.tyMotionStd1.tyNumNomSpd.diValue;
				eMagAWOpen2Act	:= MagAWActGoWidth;

				IF p_eMagAWOpen2Stat = MagAWActGoWidth AND p_eMagAWOpen2Status = Done THEN
					eMagAWOpen2Act	:= MagAWActIdle;
					usiMagAWSelfTestStep1 := 30;
				END_IF

			30:
				eMag2AWEngageAct	:= PneuActSetRet;

				IF p_eMag2AWEngageStat = PneuActSetRet AND p_eMag2AWEngageStatus = Done THEN
					eMag2AWEngageAct	:= PneuActIdle;
					usiMagAWSelfTestStep1 := 40;
				END_IF

			40:
				fbMagAWSelfTestTim1(IN:= TRUE);
				IF fbMagAWSelfTestTim1.Q THEN
					usiMagAWSelfTestStep1 := 0;
					fbMagAWSelfTestTim1(IN:= FALSE);
				END_IF
		END_CASE
	END_IF

END_ACTION
```

#### Act_OptP0938FBCtrl3.st
```iecst
ACTION Act_OptP0938FBCtrl3:

	//Motor
	fbJogSlowToFastDlyTm.PT	:= T#2s;
	fbJogSlowToFastDlyTm;
	fbLmtRstTm;

	IF EDGENEG(bMagAWSelfTest) THEN
		eMag3AWEngageAct	:= PneuActIdle;
		eMagAWOpen3Act	:= MagAWActIdle;
	END_IF

	IF bMagAWSelfTest = FALSE THEN
		usiMagAWSelfTestStep2 := 0;
		//Interruption
		IF tyP0938MagAW.tyMagAW3.tyBtnMtrGearEngage.bRtCompl = TRUE AND (EDGENEG(p_tyDI.bMagPresentSen3) OR EDGEPOS(p_eMag3AWEngageStatus = Error)) THEN
			tyP0938MagAW.tyMotionStd3.tyBtnStop.bRtCompl	:= TRUE;
		END_IF

		IF EDGEPOS((p_udiMagAWOpen3AxisErrID = 21570 OR p_udiMagAWOpen3AxisErrID = 21571) AND tyP0938MagAW.tyMotionStd3.tyBtnJogOpen.bValue = FALSE AND tyP0938MagAW.tyMotionStd3.tyBtnJogClose.bValue = FALSE) THEN
			fbLmtRstTm.IN	:= TRUE;
		END_IF

		IF fbLmtRstTm.Q = TRUE THEN
			tyP0938MagAW.tyMotionStd3.tyBtnRst.bRtCompl		:= TRUE;
		END_IF

		IF (tyP0938MagAW.tyMotionStd3.tyBtnJogOpen.bValue = FALSE AND tyP0938MagAW.tyMotionStd3.tyBtnJogClose.bValue = FALSE) AND (p_bMagAWOpen3Jogging = TRUE) THEN
			bJogStopMagAW3	:= TRUE;
		END_IF

		IF tyP0938MagAW.tyMotionStd3.tyBtnStop.bRtCompl = TRUE THEN

			IF tyP0938MagAW.tyMagAW3.tyBtnMtrGearEngage.bRtCompl = TRUE THEN
				eMagAWOpen3Act		:= MagAWActEngageStop;
				eMag3AWEngageAct	:= PneuActIdle;
			ELSE
				eMagAWOpen3Act		:= MagAWActStop;
			END_IF

			IF (p_eMagAWOpen3Stat = MagAWActStop AND p_eMagAWOpen3Status = Done) OR (p_eMagAWOpen3Stat = MagAWActEngageStop AND p_eMagAWOpen3Status = Done) THEN
				eMagAWOpen3Act	:= MagAWActIdle;

				tyP0938MagAW.tyMotionStd3.tyBtnStop.bRtCompl		:= FALSE;
				tyP0938MagAW.tyMotionStd3.tyBtnJogOpen.bRtCompl		:= FALSE;
				tyP0938MagAW.tyMotionStd3.tyBtnJogClose.bRtCompl	:= FALSE;
				tyP0938MagAW.tyMotionStd3.tyBtnOrigin.bRtCompl		:= FALSE;
				tyP0938MagAW.tyMotionStd3.tyBtnMovAbs.bRtCompl		:= FALSE;
				tyP0938MagAW.tyMotionStd3.tyBtnMovRel.bRtCompl		:= FALSE;
				tyP0938MagAW.tyMagAW3.tyBtnGo.bRtCompl				:= FALSE;
				tyP0938MagAW.tyMagAW3.tyBtnMtrGearEngage.bRtCompl	:= FALSE;

				tyP0938MagAW.tyMotionStd3.tyBtnStop.bValue			:= TRUE;
				tyP0938MagAW.tyMotionStd3.tyBtnJogOpen.bValue		:= FALSE;
				tyP0938MagAW.tyMotionStd3.tyBtnJogClose.bValue		:= FALSE;
				tyP0938MagAW.tyMotionStd3.tyBtnOrigin.bValue		:= FALSE;
				tyP0938MagAW.tyMotionStd3.tyBtnMovAbs.bValue		:= FALSE;
				tyP0938MagAW.tyMotionStd3.tyBtnMovRel.bValue		:= FALSE;
				tyP0938MagAW.tyMagAW3.tyBtnGo.bValue				:= FALSE;
				tyP0938MagAW.tyMagAW3.tyBtnMtrGearEngage.bValue		:= FALSE;

				tyP0938MagAW.tyMotionStd3.tyBtnStop.bRtLk			:= TRUE;
				tyP0938MagAW.tyMotionStd3.tyBtnJogOpen.bRtLk		:= FALSE;
				tyP0938MagAW.tyMotionStd3.tyBtnJogClose.bRtLk		:= FALSE;
				tyP0938MagAW.tyMotionStd3.tyBtnOrigin.bRtLk			:= FALSE;
				tyP0938MagAW.tyMotionStd3.tyBtnMovAbs.bRtLk			:= FALSE;
				tyP0938MagAW.tyMotionStd3.tyBtnMovRel.bRtLk			:= FALSE;
				tyP0938MagAW.tyMagAW3.tyBtnGo.bRtLk					:= FALSE;
				tyP0938MagAW.tyMagAW3.tyBtnMtrGearEngage.bRtLk		:= FALSE;
			END_IF

		ELSIF (tyP0938MagAW.tyMotionStd3.tyBtnJogOpen.bRtCompl = TRUE) OR (tyP0938MagAW.tyMotionStd3.tyBtnJogClose.bRtCompl = TRUE) OR (bJogStopMagAW3 = TRUE) THEN
			bJogSlow					:= FALSE;
			bJogFast					:= FALSE;
			fbJogSlowToFastDlyTm.IN		:= FALSE;

			eMagAWOpen3Act	:= MagAWActJogStop;

			IF p_eMagAWOpen3Stat = MagAWActJogStop AND p_eMagAWOpen3Status = Done THEN
				eMagAWOpen3Act	:= MagAWActIdle;

				bJogStopMagAW3	:= FALSE;

				tyP0938MagAW.tyMotionStd3.tyBtnStop.bRtCompl		:= FALSE;
				tyP0938MagAW.tyMotionStd3.tyBtnJogOpen.bRtCompl		:= FALSE;
				tyP0938MagAW.tyMotionStd3.tyBtnJogClose.bRtCompl	:= FALSE;
				tyP0938MagAW.tyMotionStd3.tyBtnOrigin.bRtCompl		:= FALSE;
				tyP0938MagAW.tyMotionStd3.tyBtnMovAbs.bRtCompl		:= FALSE;
				tyP0938MagAW.tyMotionStd3.tyBtnMovRel.bRtCompl		:= FALSE;
				tyP0938MagAW.tyMagAW3.tyBtnGo.bRtCompl				:= FALSE;

				tyP0938MagAW.tyMotionStd3.tyBtnStop.bValue			:= TRUE;
				tyP0938MagAW.tyMotionStd3.tyBtnJogOpen.bValue		:= FALSE;
				tyP0938MagAW.tyMotionStd3.tyBtnJogClose.bValue		:= FALSE;
				tyP0938MagAW.tyMotionStd3.tyBtnOrigin.bValue		:= FALSE;
				tyP0938MagAW.tyMotionStd3.tyBtnMovAbs.bValue		:= FALSE;
				tyP0938MagAW.tyMotionStd3.tyBtnMovRel.bValue		:= FALSE;
				tyP0938MagAW.tyMagAW3.tyBtnGo.bValue				:= FALSE;

				tyP0938MagAW.tyMotionStd3.tyBtnStop.bRtLk			:= TRUE;
				tyP0938MagAW.tyMotionStd3.tyBtnJogOpen.bRtLk		:= FALSE;
				tyP0938MagAW.tyMotionStd3.tyBtnJogClose.bRtLk		:= FALSE;
				tyP0938MagAW.tyMotionStd3.tyBtnOrigin.bRtLk			:= FALSE;
				tyP0938MagAW.tyMotionStd3.tyBtnMovAbs.bRtLk			:= FALSE;
				tyP0938MagAW.tyMotionStd3.tyBtnMovRel.bRtLk			:= FALSE;
				tyP0938MagAW.tyMagAW3.tyBtnGo.bRtLk					:= FALSE;
			END_IF

		ELSIF tyP0938MagAW.tyMotionStd3.tyBtnPwr.bRtCompl = TRUE THEN
			tyP0938MagAW.tyMotionStd3.tyBtnPwr.bRtLk	:= TRUE;

			IF tyP0938MagAW.tyMotionStd3.tyBtnPwr.bValue = TRUE THEN
				eMagAWOpen3Act	:= MagAWActPwrOn;

				IF p_eMagAWOpen3Stat = MagAWActPwrOn AND p_eMagAWOpen3Status = Done THEN
					eMagAWOpen3Act	:= MagAWActIdle;

					tyP0938MagAW.tyMotionStd3.tyBtnPwr.bRtCompl	:= FALSE;
					tyP0938MagAW.tyMotionStd3.tyBtnPwr.bRtLk	:= FALSE;
				END_IF
			ELSE
				eMagAWOpen3Act	:= MagAWActPwrOff;

				IF p_eMagAWOpen3Stat = MagAWActPwrOff AND p_eMagAWOpen3Status = Done THEN
					eMagAWOpen3Act	:= MagAWActIdle;

					tyP0938MagAW.tyMotionStd3.tyBtnPwr.bRtCompl	:= FALSE;
					tyP0938MagAW.tyMotionStd3.tyBtnPwr.bRtLk	:= FALSE;
				END_IF
			END_IF

		ELSIF tyP0938MagAW.tyMotionStd3.tyBtnOrigin.bRtCompl = TRUE THEN
			tyP0938MagAW.tyMotionStd3.tyBtnOrigin.bValue	:= TRUE;
			tyP0938MagAW.tyMotionStd3.tyBtnStop.bValue		:= FALSE;

			tyP0938MagAW.tyMotionStd3.tyBtnOrigin.bRtLk		:= TRUE;
			tyP0938MagAW.tyMotionStd3.tyBtnStop.bRtLk		:= FALSE;

			eMagAWOpen3Act	:= MagAWActHoming;

			IF p_eMagAWOpen3Stat = MagAWActHoming AND p_eMagAWOpen3Status = Done THEN
				eMagAWOpen3Act	:= MagAWActIdle;

				tyP0938MagAW.tyMotionStd3.tyBtnOrigin.bRtCompl	:= FALSE;
				tyP0938MagAW.tyMotionStd3.tyBtnOrigin.bValue	:= FALSE;
				tyP0938MagAW.tyMotionStd3.tyBtnStop.bValue		:= TRUE;

				tyP0938MagAW.tyMotionStd3.tyBtnOrigin.bRtLk		:= FALSE;
				tyP0938MagAW.tyMotionStd3.tyBtnStop.bRtLk		:= TRUE;
			END_IF

		ELSIF tyP0938MagAW.tyMotionStd3.tyBtnRst.bRtCompl = TRUE THEN
			tyP0938MagAW.tyMotionStd3.tyBtnRst.bValue	:= TRUE;
			tyP0938MagAW.tyMotionStd3.tyBtnRst.bRtLk	:= TRUE;

			eMagAWOpen3Act	:= MagAWActRstAxisErr;

			IF p_eMagAWOpen3Stat = MagAWActRstAxisErr AND p_eMagAWOpen3Status = Done THEN
				eMagAWOpen3Act	:= MagAWActIdle;

				tyP0938MagAW.tyMotionStd3.tyBtnRst.bRtCompl	:= FALSE;
				tyP0938MagAW.tyMotionStd3.tyBtnRst.bValue	:= FALSE;
				tyP0938MagAW.tyMotionStd3.tyBtnRst.bRtLk	:= FALSE;

				fbLmtRstTm.IN	:= FALSE;
			END_IF

		ELSIF tyP0938MagAW.tyMagAW3.tyBtnGo.bRtCompl = TRUE THEN
			tyP0938MagAW.tyMagAW3.tyBtnGo.bValue		:= TRUE;
			tyP0938MagAW.tyMotionStd3.tyBtnStop.bValue	:= FALSE;

			tyP0938MagAW.tyMagAW3.tyBtnGo.bRtLk			:= TRUE;
			tyP0938MagAW.tyMotionStd3.tyBtnStop.bRtLk	:= FALSE;

			diMnlMagAW3GoWidth	:= tyP0938MagAW.tyMagAW3.tyNumNewWidth.diValue;
			diMnlMagAW3NomSpd	:= tyP0938MagAW.tyMotionStd3.tyNumNomSpd.diValue;

			eMagAWOpen3Act	:= MagAWActGoWidth;

			IF p_eMagAWOpen3Stat = MagAWActGoWidth AND p_eMagAWOpen3Status = Done THEN
				eMagAWOpen3Act	:= MagAWActIdle;

				tyP0938MagAW.tyMagAW3.tyBtnGo.bRtCompl		:= FALSE;
				tyP0938MagAW.tyMagAW3.tyBtnGo.bValue		:= FALSE;
				tyP0938MagAW.tyMotionStd3.tyBtnStop.bValue	:= TRUE;

				tyP0938MagAW.tyMagAW3.tyBtnGo.bRtLk			:= FALSE;
				tyP0938MagAW.tyMotionStd3.tyBtnStop.bRtLk	:= TRUE;
			END_IF

		ELSIF tyP0938MagAW.tyMotionStd3.tyBtnMovAbs.bRtCompl = TRUE THEN
			tyP0938MagAW.tyMotionStd3.tyBtnMovAbs.bValue	:= TRUE;
			tyP0938MagAW.tyMotionStd3.tyBtnStop.bValue		:= FALSE;

			tyP0938MagAW.tyMotionStd3.tyBtnMovAbs.bRtLk		:= TRUE;
			tyP0938MagAW.tyMotionStd3.tyBtnStop.bRtLk		:= FALSE;

			diMnlMagAW3TargetPos	:= tyP0938MagAW.tyMotionStd3.tyNumTargetPos.diValue;
			diMnlMagAW3NomSpd		:= tyP0938MagAW.tyMotionStd3.tyNumNomSpd.diValue;

			eMagAWOpen3Act	:= MagAWActMovAbs;

			IF p_eMagAWOpen3Stat = MagAWActMovAbs AND p_eMagAWOpen3Status = Done THEN
				eMagAWOpen3Act	:= MagAWActIdle;

				tyP0938MagAW.tyMotionStd3.tyBtnMovAbs.bRtCompl	:= FALSE;
				tyP0938MagAW.tyMotionStd3.tyBtnMovAbs.bValue	:= FALSE;
				tyP0938MagAW.tyMotionStd3.tyBtnStop.bValue		:= TRUE;

				tyP0938MagAW.tyMotionStd3.tyBtnMovAbs.bRtLk		:= FALSE;
				tyP0938MagAW.tyMotionStd3.tyBtnStop.bRtLk		:= TRUE;
			END_IF

		ELSIF tyP0938MagAW.tyMotionStd3.tyBtnMovRel.bRtCompl = TRUE THEN
			tyP0938MagAW.tyMotionStd3.tyBtnMovRel.bValue	:= TRUE;
			tyP0938MagAW.tyMotionStd3.tyBtnStop.bValue		:= FALSE;

			tyP0938MagAW.tyMotionStd3.tyBtnMovRel.bRtLk		:= TRUE;
			tyP0938MagAW.tyMotionStd3.tyBtnStop.bRtLk		:= FALSE;

			diMnlMagAW3StepSize	:= tyP0938MagAW.tyMotionStd3.tyNumStepSize.diValue;
			diMnlMagAW3NomSpd	:= tyP0938MagAW.tyMotionStd3.tyNumNomSpd.diValue;

			eMagAWOpen3Act	:= MagAWActMovRel;

			IF p_eMagAWOpen3Stat = MagAWActMovRel AND p_eMagAWOpen3Status = Done THEN
				eMagAWOpen3Act	:= MagAWActIdle;

				tyP0938MagAW.tyMotionStd3.tyBtnMovRel.bRtCompl	:= FALSE;
				tyP0938MagAW.tyMotionStd3.tyBtnMovRel.bValue	:= FALSE;
				tyP0938MagAW.tyMotionStd3.tyBtnStop.bValue		:= TRUE;

				tyP0938MagAW.tyMotionStd3.tyBtnMovRel.bRtLk		:= FALSE;
				tyP0938MagAW.tyMotionStd3.tyBtnStop.bRtLk		:= TRUE;
			END_IF

		ELSIF (tyP0938MagAW.tyMotionStd3.tyBtnJogOpen.bValue = TRUE) AND (fbJogSlowToFastDlyTm.Q = FALSE) AND (bJogSlow = FALSE) THEN
			tyP0938MagAW.tyMotionStd3.tyBtnStop.bValue	:= FALSE;
			tyP0938MagAW.tyMotionStd3.tyBtnStop.bRtLk	:= FALSE;

			fbJogSlowToFastDlyTm.IN	:= TRUE;

			diMnlMagAW3JogSpd	:= tyP0938MagAW.tyMotionStd3.tyNumSlwSpd.diValue;

			eMagAWOpen3Act	:= MagAWActJogOpen;

			IF p_eMagAWOpen3Stat = MagAWActJogOpen AND p_eMagAWOpen3Status = Done THEN
				eMagAWOpen3Act				:= MagAWActIdle;
				bJogSlow				:= TRUE;
			ELSIF p_eMagAWOpen3Status = Error THEN
				fbJogSlowToFastDlyTm.IN	:= FALSE;
				bJogSlow				:= TRUE;
			END_IF

		ELSIF (tyP0938MagAW.tyMotionStd3.tyBtnJogOpen.bValue = TRUE) AND (fbJogSlowToFastDlyTm.Q = TRUE) AND (bJogFast = FALSE) THEN
			tyP0938MagAW.tyMotionStd3.tyBtnStop.bValue	:= FALSE;
			tyP0938MagAW.tyMotionStd3.tyBtnStop.bRtLk	:= FALSE;

			fbJogSlowToFastDlyTm.IN	:= TRUE;

			diMnlMagAW3JogSpd	:= tyP0938MagAW.tyMotionStd3.tyNumNomSpd.diValue;

			eMagAWOpen3Act	:= MagAWActJogOpen;

			IF p_eMagAWOpen3Stat = MagAWActJogOpen AND p_eMagAWOpen3Status = Done THEN
				eMagAWOpen3Act				:= MagAWActIdle;
				bJogFast				:= TRUE;
			ELSIF p_eMagAWOpen3Status = Error THEN
				fbJogSlowToFastDlyTm.IN	:= FALSE;
				bJogFast				:= TRUE;
			END_IF

		ELSIF (tyP0938MagAW.tyMotionStd3.tyBtnJogClose.bValue = TRUE) AND (fbJogSlowToFastDlyTm.Q = FALSE) AND (bJogSlow = FALSE) THEN
			tyP0938MagAW.tyMotionStd3.tyBtnStop.bValue	:= FALSE;
			tyP0938MagAW.tyMotionStd3.tyBtnStop.bRtLk	:= FALSE;

			fbJogSlowToFastDlyTm.IN	:= TRUE;

			diMnlMagAW3JogSpd	:= tyP0938MagAW.tyMotionStd3.tyNumSlwSpd.diValue;

			eMagAWOpen3Act	:= MagAWActJogClose;

			IF p_eMagAWOpen3Stat = MagAWActJogClose AND p_eMagAWOpen3Status = Done THEN
				eMagAWOpen3Act				:= MagAWActIdle;
				bJogSlow				:= TRUE;
			ELSIF p_eMagAWOpen3Status = Error THEN
				fbJogSlowToFastDlyTm.IN	:= FALSE;
				bJogSlow				:= TRUE;
			END_IF

		ELSIF (tyP0938MagAW.tyMotionStd3.tyBtnJogClose.bValue = TRUE) AND (fbJogSlowToFastDlyTm.Q = TRUE) AND (bJogFast = FALSE) THEN
			tyP0938MagAW.tyMotionStd3.tyBtnStop.bValue	:= FALSE;
			tyP0938MagAW.tyMotionStd3.tyBtnStop.bRtLk	:= FALSE;

			fbJogSlowToFastDlyTm.IN	:= TRUE;

			diMnlMagAW3JogSpd	:= tyP0938MagAW.tyMotionStd3.tyNumNomSpd.diValue;

			eMagAWOpen3Act	:= MagAWActJogClose;

			IF p_eMagAWOpen3Stat = MagAWActJogClose AND p_eMagAWOpen3Status = Done THEN
				eMagAWOpen3Act				:= MagAWActIdle;
				bJogFast				:= TRUE;
			ELSIF p_eMagAWOpen3Status = Error THEN
				fbJogSlowToFastDlyTm.IN	:= FALSE;
				bJogFast				:= TRUE;
			END_IF

		ELSIF tyP0938MagAW.tyMagAW3.tyBtnMtrGearEngage.bRtCompl = TRUE THEN
			tyP0938MagAW.tyMagAW3.tyBtnMtrGearEngage.bValue	:= TRUE;
			tyP0938MagAW.tyMotionStd3.tyBtnStop.bValue		:= FALSE;

			tyP0938MagAW.tyMagAW3.tyBtnMtrGearEngage.bRtLk	:= TRUE;
			tyP0938MagAW.tyMotionStd3.tyBtnStop.bRtLk		:= FALSE;

			eMagAWOpen3Act	:= MagAWActEngage;

			IF p_bMagAWOpen3Engaging = TRUE THEN
				eMag3AWEngageAct	:= PneuActExt;

				tyP0938MagAW.tyMagAW3.tyBtnEngage.bValue	:= TRUE;
				tyP0938MagAW.tyMagAW3.tyBtnDisengage.bValue	:= FALSE;
			END_IF

			IF (p_eMagAWOpen3Stat = MagAWActEngage AND p_eMagAWOpen3Status = Done) AND (p_eMag3AWEngageStat = PneuActExt AND p_eMag3AWEngageStatus = Done) THEN
				eMagAWOpen3Act		:= MagAWActIdle;
				eMag3AWEngageAct	:= PneuActIdle;

				tyP0938MagAW.tyMagAW3.tyBtnMtrGearEngage.bRtCompl	:= FALSE;
				tyP0938MagAW.tyMagAW3.tyBtnMtrGearEngage.bValue		:= FALSE;
				tyP0938MagAW.tyMotionStd3.tyBtnStop.bValue			:= TRUE;

				tyP0938MagAW.tyMagAW3.tyBtnMtrGearEngage.bRtLk		:= FALSE;
				tyP0938MagAW.tyMotionStd3.tyBtnStop.bRtLk			:= TRUE;
			END_IF

		END_IF

		//Pneumatic
		IF p_bMag3AWEngageTwoCtrlOut = FALSE THEN

			IF tyP0938MagAW.tyMagAW3.tyBtnDisengage.bRtCompl = TRUE THEN
				tyP0938MagAW.tyMagAW3.tyBtnDisengage.bValue	:= TRUE;
				tyP0938MagAW.tyMagAW3.tyBtnEngage.bValue	:= FALSE;

				eMag3AWEngageAct	:= PneuActSetRet;

				IF p_eMag3AWEngageStat = PneuActSetRet AND p_eMag3AWEngageStatus = Done THEN
					eMag3AWEngageAct	:= PneuActIdle;

					tyP0938MagAW.tyMagAW3.tyBtnDisengage.bRtCompl	:= FALSE;
				END_IF

			ELSIF tyP0938MagAW.tyMagAW3.tyBtnEngage.bRtCompl = TRUE THEN
				tyP0938MagAW.tyMagAW3.tyBtnEngage.bValue	:= TRUE;
				tyP0938MagAW.tyMagAW3.tyBtnDisengage.bValue	:= FALSE;

				eMag3AWEngageAct	:= PneuActSetExt;

				IF p_eMag3AWEngageStat = PneuActSetExt AND p_eMag3AWEngageStatus = Done THEN
					eMag3AWEngageAct	:= PneuActIdle;

					tyP0938MagAW.tyMagAW3.tyBtnEngage.bRtCompl	:= FALSE;
				END_IF

			END_IF

		ELSE

			IF (tyP0938MagAW.tyMagAW3.tyBtnDisengage.bRtCompl = TRUE) OR (tyP0938MagAW.tyMagAW3.tyBtnEngage.bRtCompl = TRUE) THEN

				IF (tyP0938MagAW.tyMagAW3.tyBtnDisengage.bValue = TRUE) AND (tyP0938MagAW.tyMagAW3.tyBtnEngage.bValue = TRUE) THEN
					eMag3AWEngageAct	:= PneuActSetAll;

					IF p_eMag3AWEngageStat = PneuActSetAll AND p_eMag3AWEngageStatus = Done THEN
						eMag3AWEngageAct	:= PneuActIdle;

						tyP0938MagAW.tyMagAW3.tyBtnDisengage.bRtCompl	:= FALSE;
						tyP0938MagAW.tyMagAW3.tyBtnEngage.bRtCompl		:= FALSE;
					END_IF

				ELSIF (tyP0938MagAW.tyMagAW3.tyBtnDisengage.bValue = TRUE) AND (tyP0938MagAW.tyMagAW3.tyBtnEngage.bValue = FALSE) THEN
					eMag3AWEngageAct	:= PneuActSetRet;

					IF p_eMag3AWEngageStat = PneuActSetRet AND p_eMag3AWEngageStatus = Done THEN
						eMag3AWEngageAct	:= PneuActIdle;

						tyP0938MagAW.tyMagAW3.tyBtnDisengage.bRtCompl	:= FALSE;
						tyP0938MagAW.tyMagAW3.tyBtnEngage.bRtCompl		:= FALSE;
					END_IF

				ELSIF (tyP0938MagAW.tyMagAW3.tyBtnDisengage.bValue = FALSE) AND (tyP0938MagAW.tyMagAW3.tyBtnEngage.bValue = TRUE) THEN
					eMag3AWEngageAct	:= PneuActSetExt;

					IF p_eMag3AWEngageStat = PneuActSetExt AND p_eMag3AWEngageStatus = Done THEN
						eMag3AWEngageAct	:= PneuActIdle;

						tyP0938MagAW.tyMagAW3.tyBtnDisengage.bRtCompl	:= FALSE;
						tyP0938MagAW.tyMagAW3.tyBtnEngage.bRtCompl		:= FALSE;
					END_IF

				ELSE
					eMag3AWEngageAct	:= PneuActRstAll;

					IF p_eMag3AWEngageStat = PneuActRstAll AND p_eMag3AWEngageStatus = Done THEN
						eMag3AWEngageAct	:= PneuActIdle;

						tyP0938MagAW.tyMagAW3.tyBtnDisengage.bRtCompl	:= FALSE;
						tyP0938MagAW.tyMagAW3.tyBtnEngage.bRtCompl		:= FALSE;
					END_IF

				END_IF

			END_IF

		END_IF

	ELSE
		CASE usiMagAWSelfTestStep2 OF

			0: IF p_bMagConv2Clp3ClprFixClampCtrl THEN

					eMagAWOpen3Act	:= MagAWActEngage;

					eMag3AWEngageAct	:= PneuActExt;

					IF (p_eMagAWOpen3Stat = MagAWActEngage AND p_eMagAWOpen3Status = Done)
						AND (p_eMag3AWEngageStat = PneuActExt AND p_eMag3AWEngageStatus = Done)
						THEN
						eMagAWOpen3Act		:= MagAWActIdle;
						eMag3AWEngageAct	:= PneuActIdle;
						usiMagAWSelfTestStep2 := 10;
					END_IF

				END_IF

			10:
				eMagAWOpen3Act	:= MagAWActHoming;

				IF p_eMagAWOpen3Stat = MagAWActHoming AND p_eMagAWOpen3Status = Done THEN
					eMagAWOpen3Act	:= MagAWActIdle;
					usiMagAWSelfTestStep2 := 20;
				END_IF

			20:

				diMnlMagAW3GoWidth	:= tyP0938MagAW.tyMagAW1.tyNumNewWidth.diValue;
				diMnlMagAW3NomSpd		:= tyP0938MagAW.tyMotionStd1.tyNumNomSpd.diValue;
				eMagAWOpen3Act	:= MagAWActGoWidth;

				IF p_eMagAWOpen3Stat = MagAWActGoWidth AND p_eMagAWOpen3Status = Done THEN
					eMagAWOpen3Act	:= MagAWActIdle;
					usiMagAWSelfTestStep2 := 30;
				END_IF

			30:
				eMag3AWEngageAct	:= PneuActSetRet;

				IF p_eMag3AWEngageStat = PneuActSetRet AND p_eMag3AWEngageStatus = Done THEN
					eMag3AWEngageAct	:= PneuActIdle;
					usiMagAWSelfTestStep2 := 40;
				END_IF

			40:
				fbMagAWSelfTestTim2(IN:= TRUE);
				IF fbMagAWSelfTestTim2.Q THEN
					usiMagAWSelfTestStep2 := 0;
					fbMagAWSelfTestTim2(IN:= FALSE);
				END_IF
		END_CASE
	END_IF

END_ACTION
```

#### Act_OptP0938FBStat.st
```iecst
ACTION Act_OptP0938FBStat:

	(*Magazine Auto Width 1*)
	IF p_bMagAWOpen1AxisErr = TRUE THEN
		tyP0938MagAW.tyMotionStd1.tyStringStat.sValue	:= p_sMagAWOpen1AxisErrTxt;
	ELSE
		tyP0938MagAW.tyMotionStd1.tyStringStat.sValue	:= p_sMagAWOpen1StatTxt;
	END_IF

	(*Magazine Auto Width 2*)
	IF p_bMagAWOpen2AxisErr = TRUE THEN
		tyP0938MagAW.tyMotionStd2.tyStringStat.sValue	:= p_sMagAWOpen2AxisErrTxt;
	ELSE
		tyP0938MagAW.tyMotionStd2.tyStringStat.sValue	:= p_sMagAWOpen2StatTxt;
	END_IF

	(*Magazine Auto Width 3*)
	IF p_bMagAWOpen3AxisErr = TRUE THEN
		tyP0938MagAW.tyMotionStd3.tyStringStat.sValue	:= p_sMagAWOpen3AxisErrTxt;
	ELSE
		tyP0938MagAW.tyMotionStd3.tyStringStat.sValue	:= p_sMagAWOpen3StatTxt;
	END_IF

END_ACTION
```

#### Act_OptP0938Mask.st
```iecst
ACTION Act_OptP0938Mask:

	(*Magazine Auto Width 1*)
	//Interlock Power
	IF p_bMagAWOpen1AxisErr = TRUE AND p_bMagAWOpen1PwrOn = FALSE THEN
		fUIInRtStatOff(ADR(tyP0938MagAW.tyMotionStd1.tyBtnPwr.uiMaskRtStat));
		tyP0938MagAW.tyMotionStd1.tyBtnPwr.bValue	:= FALSE;
	ELSE
		fUIInRtStatHide(ADR(tyP0938MagAW.tyMotionStd1.tyBtnPwr.uiMaskRtStat));
	END_IF

	//Interlock Others Move
	IF p_bMagAWOpen1AxisErr = TRUE OR p_bMagAWOpen1PwrOn = FALSE THEN
		fUIInRtStatOff(ADR(tyP0938MagAW.tyMotionStd1.tyBtnOrigin.uiMaskRtStat));
		fUIInRtStatOff(ADR(tyP0938MagAW.tyMotionStd1.tyBtnMovRel.uiMaskRtStat));
		fUIInRtStatOff(ADR(tyP0938MagAW.tyMotionStd1.tyBtnJogOpen.uiMaskRtStat));
		fUIInRtStatOff(ADR(tyP0938MagAW.tyMotionStd1.tyBtnJogClose.uiMaskRtStat));
	ELSE
		fUIInRtStatHide(ADR(tyP0938MagAW.tyMotionStd1.tyBtnOrigin.uiMaskRtStat));
		fUIInRtStatHide(ADR(tyP0938MagAW.tyMotionStd1.tyBtnMovRel.uiMaskRtStat));
		fUIInRtStatHide(ADR(tyP0938MagAW.tyMotionStd1.tyBtnJogOpen.uiMaskRtStat));
		fUIInRtStatHide(ADR(tyP0938MagAW.tyMotionStd1.tyBtnJogClose.uiMaskRtStat));
	END_IF

	//Interlock Move Absolute
	IF p_bMagAWOpen1AxisErr = TRUE OR p_bMagAWOpen1PwrOn = FALSE OR p_bMagAWOpen1IsHomed = FALSE THEN
		fUIInRtStatOff(ADR(tyP0938MagAW.tyMagAW1.tyBtnGo.uiMaskRtStat));
		fUIInRtStatOff(ADR(tyP0938MagAW.tyMotionStd1.tyBtnMovAbs.uiMaskRtStat));
	ELSE
		fUIInRtStatHide(ADR(tyP0938MagAW.tyMagAW1.tyBtnGo.uiMaskRtStat));
		fUIInRtStatHide(ADR(tyP0938MagAW.tyMotionStd1.tyBtnMovAbs.uiMaskRtStat));
	END_IF

	//Engage
	IF p_bMagAWOpen1AxisErr = TRUE OR p_bMagAWOpen1PwrOn = FALSE OR p_tyDI.bMagPresentSen1 = FALSE OR tyP0938MagAW.tyMagAW1.tyBtnEngageRS.bValue = TRUE OR tyP0938MagAW.tyMagAW1.tyBtnEngage.bRtCompl = TRUE OR tyP0938MagAW.tyMagAW1.tyBtnDisengage.bRtCompl = TRUE OR p_eMag1AWEngageStatus = Error THEN
		fUIInRtStatOff(ADR(tyP0938MagAW.tyMagAW1.tyBtnMtrGearEngage.uiMaskRtStat));
	ELSE
		fUIInRtStatHide(ADR(tyP0938MagAW.tyMagAW1.tyBtnMtrGearEngage.uiMaskRtStat));
	END_IF

	//Interlock Limit Sensor
	IF tyP0938MagAW.tyMotionStd1.tyBtnOpenLmtSen.bValue = TRUE THEN
		fUIInRtStatOff(ADR(tyP0938MagAW.tyMotionStd1.tyBtnJogOpen.uiMaskRtStat));
	END_IF

	IF tyP0938MagAW.tyMotionStd1.tyBtnCloseLmtSen.bValue = TRUE THEN
		fUIInRtStatOff(ADR(tyP0938MagAW.tyMotionStd1.tyBtnJogClose.uiMaskRtStat));
	END_IF

	//Interlock When Moving
	IF tyP0938MagAW.tyMotionStd1.tyBtnOrigin.bRtCompl = TRUE THEN
		fUIInRtStatOff(ADR(tyP0938MagAW.tyMotionStd1.tyBtnMovAbs.uiMaskRtStat));
		fUIInRtStatOff(ADR(tyP0938MagAW.tyMotionStd1.tyBtnMovRel.uiMaskRtStat));
		fUIInRtStatOff(ADR(tyP0938MagAW.tyMotionStd1.tyBtnJogOpen.uiMaskRtStat));
		fUIInRtStatOff(ADR(tyP0938MagAW.tyMotionStd1.tyBtnJogClose.uiMaskRtStat));
		fUIInRtStatOff(ADR(tyP0938MagAW.tyMagAW1.tyBtnGo.uiMaskRtStat));
		fUIInRtStatOff(ADR(tyP0938MagAW.tyMagAW1.tyBtnMtrGearEngage.uiMaskRtStat));

	ELSIF tyP0938MagAW.tyMotionStd1.tyBtnMovAbs.bRtCompl = TRUE THEN
		fUIInRtStatOff(ADR(tyP0938MagAW.tyMotionStd1.tyBtnOrigin.uiMaskRtStat));
		fUIInRtStatOff(ADR(tyP0938MagAW.tyMotionStd1.tyBtnMovRel.uiMaskRtStat));
		fUIInRtStatOff(ADR(tyP0938MagAW.tyMotionStd1.tyBtnJogOpen.uiMaskRtStat));
		fUIInRtStatOff(ADR(tyP0938MagAW.tyMotionStd1.tyBtnJogClose.uiMaskRtStat));
		fUIInRtStatOff(ADR(tyP0938MagAW.tyMagAW1.tyBtnGo.uiMaskRtStat));
		fUIInRtStatOff(ADR(tyP0938MagAW.tyMagAW1.tyBtnMtrGearEngage.uiMaskRtStat));

	ELSIF tyP0938MagAW.tyMotionStd1.tyBtnMovRel.bRtCompl = TRUE THEN
		fUIInRtStatOff(ADR(tyP0938MagAW.tyMotionStd1.tyBtnOrigin.uiMaskRtStat));
		fUIInRtStatOff(ADR(tyP0938MagAW.tyMotionStd1.tyBtnMovAbs.uiMaskRtStat));
		fUIInRtStatOff(ADR(tyP0938MagAW.tyMotionStd1.tyBtnJogOpen.uiMaskRtStat));
		fUIInRtStatOff(ADR(tyP0938MagAW.tyMotionStd1.tyBtnJogClose.uiMaskRtStat));
		fUIInRtStatOff(ADR(tyP0938MagAW.tyMagAW1.tyBtnGo.uiMaskRtStat));
		fUIInRtStatOff(ADR(tyP0938MagAW.tyMagAW1.tyBtnMtrGearEngage.uiMaskRtStat));

	ELSIF tyP0938MagAW.tyMotionStd1.tyBtnJogOpen.bRtCompl = TRUE OR tyP0938MagAW.tyMotionStd1.tyBtnJogOpen.bValue = TRUE THEN
		fUIInRtStatOff(ADR(tyP0938MagAW.tyMotionStd1.tyBtnOrigin.uiMaskRtStat));
		fUIInRtStatOff(ADR(tyP0938MagAW.tyMotionStd1.tyBtnMovAbs.uiMaskRtStat));
		fUIInRtStatOff(ADR(tyP0938MagAW.tyMotionStd1.tyBtnMovRel.uiMaskRtStat));
		fUIInRtStatOff(ADR(tyP0938MagAW.tyMotionStd1.tyBtnJogClose.uiMaskRtStat));
		fUIInRtStatOff(ADR(tyP0938MagAW.tyMagAW1.tyBtnGo.uiMaskRtStat));
		fUIInRtStatOff(ADR(tyP0938MagAW.tyMagAW1.tyBtnMtrGearEngage.uiMaskRtStat));

	ELSIF tyP0938MagAW.tyMotionStd1.tyBtnJogClose.bRtCompl = TRUE OR tyP0938MagAW.tyMotionStd1.tyBtnJogClose.bValue = TRUE THEN
		fUIInRtStatOff(ADR(tyP0938MagAW.tyMotionStd1.tyBtnOrigin.uiMaskRtStat));
		fUIInRtStatOff(ADR(tyP0938MagAW.tyMotionStd1.tyBtnMovAbs.uiMaskRtStat));
		fUIInRtStatOff(ADR(tyP0938MagAW.tyMotionStd1.tyBtnMovRel.uiMaskRtStat));
		fUIInRtStatOff(ADR(tyP0938MagAW.tyMotionStd1.tyBtnJogOpen.uiMaskRtStat));
		fUIInRtStatOff(ADR(tyP0938MagAW.tyMagAW1.tyBtnGo.uiMaskRtStat));
		fUIInRtStatOff(ADR(tyP0938MagAW.tyMagAW1.tyBtnMtrGearEngage.uiMaskRtStat));

	ELSIF tyP0938MagAW.tyMagAW1.tyBtnGo.bRtCompl = TRUE THEN
		fUIInRtStatOff(ADR(tyP0938MagAW.tyMotionStd1.tyBtnOrigin.uiMaskRtStat));
		fUIInRtStatOff(ADR(tyP0938MagAW.tyMotionStd1.tyBtnMovAbs.uiMaskRtStat));
		fUIInRtStatOff(ADR(tyP0938MagAW.tyMotionStd1.tyBtnMovRel.uiMaskRtStat));
		fUIInRtStatOff(ADR(tyP0938MagAW.tyMotionStd1.tyBtnJogOpen.uiMaskRtStat));
		fUIInRtStatOff(ADR(tyP0938MagAW.tyMotionStd1.tyBtnJogClose.uiMaskRtStat));
		fUIInRtStatOff(ADR(tyP0938MagAW.tyMagAW1.tyBtnMtrGearEngage.uiMaskRtStat));

	ELSIF tyP0938MagAW.tyMagAW1.tyBtnMtrGearEngage.bRtCompl = TRUE THEN
		fUIInRtStatOff(ADR(tyP0938MagAW.tyMotionStd1.tyBtnOrigin.uiMaskRtStat));
		fUIInRtStatOff(ADR(tyP0938MagAW.tyMotionStd1.tyBtnMovAbs.uiMaskRtStat));
		fUIInRtStatOff(ADR(tyP0938MagAW.tyMotionStd1.tyBtnMovRel.uiMaskRtStat));
		fUIInRtStatOff(ADR(tyP0938MagAW.tyMotionStd1.tyBtnJogOpen.uiMaskRtStat));
		fUIInRtStatOff(ADR(tyP0938MagAW.tyMotionStd1.tyBtnJogClose.uiMaskRtStat));
		fUIInRtStatOff(ADR(tyP0938MagAW.tyMagAW1.tyBtnGo.uiMaskRtStat));

	END_IF

	//Axis Error
	IF tyP0938MagAW.tyMotionStd1.tyBtnPwr.bRtCompl = TRUE THEN
		fUIInRtStatOff(ADR(tyP0938MagAW.tyMotionStd1.tyBtnRst.uiMaskRtStat));
	ELSE
		fUIInRtStatHide(ADR(tyP0938MagAW.tyMotionStd1.tyBtnRst.uiMaskRtStat));
	END_IF

	//Pneumatic
	IF tyP0938MagAW.tyMagAW1.tyBtnMtrGearEngage.bRtCompl = TRUE THEN
		fUIInRtStatOff(ADR(tyP0938MagAW.tyMagAW1.tyBtnEngage.uiMaskRtStat));
		fUIInRtStatOff(ADR(tyP0938MagAW.tyMagAW1.tyBtnDisengage.uiMaskRtStat));
	ELSE
		fUIInRtStatHide(ADR(tyP0938MagAW.tyMagAW1.tyBtnEngage.uiMaskRtStat));
		fUIInRtStatHide(ADR(tyP0938MagAW.tyMagAW1.tyBtnDisengage.uiMaskRtStat));
	END_IF

	(*Magazine Auto Width 2*)
	//Interlock Power
	IF p_bMagAWOpen2AxisErr = TRUE AND p_bMagAWOpen2PwrOn = FALSE THEN
		fUIInRtStatOff(ADR(tyP0938MagAW.tyMotionStd2.tyBtnPwr.uiMaskRtStat));
		tyP0938MagAW.tyMotionStd2.tyBtnPwr.bValue	:= FALSE;
	ELSE
		fUIInRtStatHide(ADR(tyP0938MagAW.tyMotionStd2.tyBtnPwr.uiMaskRtStat));
	END_IF

	//Interlock Others Move
	IF p_bMagAWOpen2AxisErr = TRUE OR p_bMagAWOpen2PwrOn = FALSE THEN
		fUIInRtStatOff(ADR(tyP0938MagAW.tyMotionStd2.tyBtnOrigin.uiMaskRtStat));
		fUIInRtStatOff(ADR(tyP0938MagAW.tyMotionStd2.tyBtnMovRel.uiMaskRtStat));
		fUIInRtStatOff(ADR(tyP0938MagAW.tyMotionStd2.tyBtnJogOpen.uiMaskRtStat));
		fUIInRtStatOff(ADR(tyP0938MagAW.tyMotionStd2.tyBtnJogClose.uiMaskRtStat));
	ELSE
		fUIInRtStatHide(ADR(tyP0938MagAW.tyMotionStd2.tyBtnOrigin.uiMaskRtStat));
		fUIInRtStatHide(ADR(tyP0938MagAW.tyMotionStd2.tyBtnMovRel.uiMaskRtStat));
		fUIInRtStatHide(ADR(tyP0938MagAW.tyMotionStd2.tyBtnJogOpen.uiMaskRtStat));
		fUIInRtStatHide(ADR(tyP0938MagAW.tyMotionStd2.tyBtnJogClose.uiMaskRtStat));
	END_IF

	//Interlock Move Absolute
	IF p_bMagAWOpen2AxisErr = TRUE OR p_bMagAWOpen2PwrOn = FALSE OR p_bMagAWOpen2IsHomed = FALSE THEN
		fUIInRtStatOff(ADR(tyP0938MagAW.tyMagAW2.tyBtnGo.uiMaskRtStat));
		fUIInRtStatOff(ADR(tyP0938MagAW.tyMotionStd2.tyBtnMovAbs.uiMaskRtStat));
	ELSE
		fUIInRtStatHide(ADR(tyP0938MagAW.tyMagAW2.tyBtnGo.uiMaskRtStat));
		fUIInRtStatHide(ADR(tyP0938MagAW.tyMotionStd2.tyBtnMovAbs.uiMaskRtStat));
	END_IF

	//Engage
	IF p_bMagAWOpen2AxisErr = TRUE OR p_bMagAWOpen2PwrOn = FALSE OR p_tyDI.bMagPresentSen2 = FALSE OR tyP0938MagAW.tyMagAW2.tyBtnEngageRS.bValue = TRUE OR tyP0938MagAW.tyMagAW2.tyBtnEngage.bRtCompl = TRUE OR tyP0938MagAW.tyMagAW2.tyBtnDisengage.bRtCompl = TRUE OR p_eMag2AWEngageStatus = Error THEN
		fUIInRtStatOff(ADR(tyP0938MagAW.tyMagAW2.tyBtnMtrGearEngage.uiMaskRtStat));
	ELSE
		fUIInRtStatHide(ADR(tyP0938MagAW.tyMagAW2.tyBtnMtrGearEngage.uiMaskRtStat));
	END_IF

	//Interlock Limit Sensor
	IF tyP0938MagAW.tyMotionStd2.tyBtnOpenLmtSen.bValue = TRUE THEN
		fUIInRtStatOff(ADR(tyP0938MagAW.tyMotionStd2.tyBtnJogOpen.uiMaskRtStat));
	END_IF

	IF tyP0938MagAW.tyMotionStd2.tyBtnCloseLmtSen.bValue = TRUE THEN
		fUIInRtStatOff(ADR(tyP0938MagAW.tyMotionStd2.tyBtnJogClose.uiMaskRtStat));
	END_IF

	//Interlock When Moving
	IF tyP0938MagAW.tyMotionStd2.tyBtnOrigin.bRtCompl = TRUE THEN
		fUIInRtStatOff(ADR(tyP0938MagAW.tyMotionStd2.tyBtnMovAbs.uiMaskRtStat));
		fUIInRtStatOff(ADR(tyP0938MagAW.tyMotionStd2.tyBtnMovRel.uiMaskRtStat));
		fUIInRtStatOff(ADR(tyP0938MagAW.tyMotionStd2.tyBtnJogOpen.uiMaskRtStat));
		fUIInRtStatOff(ADR(tyP0938MagAW.tyMotionStd2.tyBtnJogClose.uiMaskRtStat));
		fUIInRtStatOff(ADR(tyP0938MagAW.tyMagAW2.tyBtnGo.uiMaskRtStat));
		fUIInRtStatOff(ADR(tyP0938MagAW.tyMagAW2.tyBtnMtrGearEngage.uiMaskRtStat));

	ELSIF tyP0938MagAW.tyMotionStd2.tyBtnMovAbs.bRtCompl = TRUE THEN
		fUIInRtStatOff(ADR(tyP0938MagAW.tyMotionStd2.tyBtnOrigin.uiMaskRtStat));
		fUIInRtStatOff(ADR(tyP0938MagAW.tyMotionStd2.tyBtnMovRel.uiMaskRtStat));
		fUIInRtStatOff(ADR(tyP0938MagAW.tyMotionStd2.tyBtnJogOpen.uiMaskRtStat));
		fUIInRtStatOff(ADR(tyP0938MagAW.tyMotionStd2.tyBtnJogClose.uiMaskRtStat));
		fUIInRtStatOff(ADR(tyP0938MagAW.tyMagAW2.tyBtnGo.uiMaskRtStat));
		fUIInRtStatOff(ADR(tyP0938MagAW.tyMagAW2.tyBtnMtrGearEngage.uiMaskRtStat));

	ELSIF tyP0938MagAW.tyMotionStd2.tyBtnMovRel.bRtCompl = TRUE THEN
		fUIInRtStatOff(ADR(tyP0938MagAW.tyMotionStd2.tyBtnOrigin.uiMaskRtStat));
		fUIInRtStatOff(ADR(tyP0938MagAW.tyMotionStd2.tyBtnMovAbs.uiMaskRtStat));
		fUIInRtStatOff(ADR(tyP0938MagAW.tyMotionStd2.tyBtnJogOpen.uiMaskRtStat));
		fUIInRtStatOff(ADR(tyP0938MagAW.tyMotionStd2.tyBtnJogClose.uiMaskRtStat));
		fUIInRtStatOff(ADR(tyP0938MagAW.tyMagAW2.tyBtnGo.uiMaskRtStat));
		fUIInRtStatOff(ADR(tyP0938MagAW.tyMagAW2.tyBtnMtrGearEngage.uiMaskRtStat));

	ELSIF tyP0938MagAW.tyMotionStd2.tyBtnJogOpen.bRtCompl = TRUE OR tyP0938MagAW.tyMotionStd2.tyBtnJogOpen.bValue = TRUE THEN
		fUIInRtStatOff(ADR(tyP0938MagAW.tyMotionStd2.tyBtnOrigin.uiMaskRtStat));
		fUIInRtStatOff(ADR(tyP0938MagAW.tyMotionStd2.tyBtnMovAbs.uiMaskRtStat));
		fUIInRtStatOff(ADR(tyP0938MagAW.tyMotionStd2.tyBtnMovRel.uiMaskRtStat));
		fUIInRtStatOff(ADR(tyP0938MagAW.tyMotionStd2.tyBtnJogClose.uiMaskRtStat));
		fUIInRtStatOff(ADR(tyP0938MagAW.tyMagAW2.tyBtnGo.uiMaskRtStat));
		fUIInRtStatOff(ADR(tyP0938MagAW.tyMagAW2.tyBtnMtrGearEngage.uiMaskRtStat));

	ELSIF tyP0938MagAW.tyMotionStd2.tyBtnJogClose.bRtCompl = TRUE OR tyP0938MagAW.tyMotionStd2.tyBtnJogClose.bValue = TRUE THEN
		fUIInRtStatOff(ADR(tyP0938MagAW.tyMotionStd2.tyBtnOrigin.uiMaskRtStat));
		fUIInRtStatOff(ADR(tyP0938MagAW.tyMotionStd2.tyBtnMovAbs.uiMaskRtStat));
		fUIInRtStatOff(ADR(tyP0938MagAW.tyMotionStd2.tyBtnMovRel.uiMaskRtStat));
		fUIInRtStatOff(ADR(tyP0938MagAW.tyMotionStd2.tyBtnJogOpen.uiMaskRtStat));
		fUIInRtStatOff(ADR(tyP0938MagAW.tyMagAW2.tyBtnGo.uiMaskRtStat));
		fUIInRtStatOff(ADR(tyP0938MagAW.tyMagAW2.tyBtnMtrGearEngage.uiMaskRtStat));

	ELSIF tyP0938MagAW.tyMagAW2.tyBtnGo.bRtCompl = TRUE THEN
		fUIInRtStatOff(ADR(tyP0938MagAW.tyMotionStd2.tyBtnOrigin.uiMaskRtStat));
		fUIInRtStatOff(ADR(tyP0938MagAW.tyMotionStd2.tyBtnMovAbs.uiMaskRtStat));
		fUIInRtStatOff(ADR(tyP0938MagAW.tyMotionStd2.tyBtnMovRel.uiMaskRtStat));
		fUIInRtStatOff(ADR(tyP0938MagAW.tyMotionStd2.tyBtnJogOpen.uiMaskRtStat));
		fUIInRtStatOff(ADR(tyP0938MagAW.tyMotionStd2.tyBtnJogClose.uiMaskRtStat));
		fUIInRtStatOff(ADR(tyP0938MagAW.tyMagAW2.tyBtnMtrGearEngage.uiMaskRtStat));

	ELSIF tyP0938MagAW.tyMagAW2.tyBtnMtrGearEngage.bRtCompl = TRUE THEN
		fUIInRtStatOff(ADR(tyP0938MagAW.tyMotionStd2.tyBtnOrigin.uiMaskRtStat));
		fUIInRtStatOff(ADR(tyP0938MagAW.tyMotionStd2.tyBtnMovAbs.uiMaskRtStat));
		fUIInRtStatOff(ADR(tyP0938MagAW.tyMotionStd2.tyBtnMovRel.uiMaskRtStat));
		fUIInRtStatOff(ADR(tyP0938MagAW.tyMotionStd2.tyBtnJogOpen.uiMaskRtStat));
		fUIInRtStatOff(ADR(tyP0938MagAW.tyMotionStd2.tyBtnJogClose.uiMaskRtStat));
		fUIInRtStatOff(ADR(tyP0938MagAW.tyMagAW2.tyBtnGo.uiMaskRtStat));

	END_IF

	//Axis Error
	IF tyP0938MagAW.tyMotionStd2.tyBtnPwr.bRtCompl = TRUE THEN
		fUIInRtStatOff(ADR(tyP0938MagAW.tyMotionStd2.tyBtnRst.uiMaskRtStat));
	ELSE
		fUIInRtStatHide(ADR(tyP0938MagAW.tyMotionStd2.tyBtnRst.uiMaskRtStat));
	END_IF

	//Pneumatic
	IF tyP0938MagAW.tyMagAW2.tyBtnMtrGearEngage.bRtCompl = TRUE THEN
		fUIInRtStatOff(ADR(tyP0938MagAW.tyMagAW2.tyBtnEngage.uiMaskRtStat));
		fUIInRtStatOff(ADR(tyP0938MagAW.tyMagAW2.tyBtnDisengage.uiMaskRtStat));
	ELSE
		fUIInRtStatHide(ADR(tyP0938MagAW.tyMagAW2.tyBtnEngage.uiMaskRtStat));
		fUIInRtStatHide(ADR(tyP0938MagAW.tyMagAW2.tyBtnDisengage.uiMaskRtStat));
	END_IF

	(*Magazine Auto Width 3*)
	//Interlock Power
	IF p_bMagAWOpen3AxisErr = TRUE AND p_bMagAWOpen3PwrOn = FALSE THEN
		fUIInRtStatOff(ADR(tyP0938MagAW.tyMotionStd3.tyBtnPwr.uiMaskRtStat));
		tyP0938MagAW.tyMotionStd3.tyBtnPwr.bValue	:= FALSE;
	ELSE
		fUIInRtStatHide(ADR(tyP0938MagAW.tyMotionStd3.tyBtnPwr.uiMaskRtStat));
	END_IF

	//Interlock Others Move
	IF p_bMagAWOpen3AxisErr = TRUE OR p_bMagAWOpen3PwrOn = FALSE THEN
		fUIInRtStatOff(ADR(tyP0938MagAW.tyMotionStd3.tyBtnOrigin.uiMaskRtStat));
		fUIInRtStatOff(ADR(tyP0938MagAW.tyMotionStd3.tyBtnMovRel.uiMaskRtStat));
		fUIInRtStatOff(ADR(tyP0938MagAW.tyMotionStd3.tyBtnJogOpen.uiMaskRtStat));
		fUIInRtStatOff(ADR(tyP0938MagAW.tyMotionStd3.tyBtnJogClose.uiMaskRtStat));
	ELSE
		fUIInRtStatHide(ADR(tyP0938MagAW.tyMotionStd3.tyBtnOrigin.uiMaskRtStat));
		fUIInRtStatHide(ADR(tyP0938MagAW.tyMotionStd3.tyBtnMovRel.uiMaskRtStat));
		fUIInRtStatHide(ADR(tyP0938MagAW.tyMotionStd3.tyBtnJogOpen.uiMaskRtStat));
		fUIInRtStatHide(ADR(tyP0938MagAW.tyMotionStd3.tyBtnJogClose.uiMaskRtStat));
	END_IF

	//Interlock Move Absolute
	IF p_bMagAWOpen3AxisErr = TRUE OR p_bMagAWOpen3PwrOn = FALSE OR p_bMagAWOpen3IsHomed = FALSE THEN
		fUIInRtStatOff(ADR(tyP0938MagAW.tyMagAW3.tyBtnGo.uiMaskRtStat));
		fUIInRtStatOff(ADR(tyP0938MagAW.tyMotionStd3.tyBtnMovAbs.uiMaskRtStat));
	ELSE
		fUIInRtStatHide(ADR(tyP0938MagAW.tyMagAW3.tyBtnGo.uiMaskRtStat));
		fUIInRtStatHide(ADR(tyP0938MagAW.tyMotionStd3.tyBtnMovAbs.uiMaskRtStat));
	END_IF

	//Engage
	IF p_bMagAWOpen3AxisErr = TRUE OR p_bMagAWOpen3PwrOn = FALSE OR p_tyDI.bMagPresentSen3 = FALSE OR tyP0938MagAW.tyMagAW3.tyBtnEngageRS.bValue = TRUE OR tyP0938MagAW.tyMagAW3.tyBtnEngage.bRtCompl = TRUE OR tyP0938MagAW.tyMagAW3.tyBtnDisengage.bRtCompl = TRUE OR p_eMag3AWEngageStatus = Error THEN
		fUIInRtStatOff(ADR(tyP0938MagAW.tyMagAW3.tyBtnMtrGearEngage.uiMaskRtStat));
	ELSE
		fUIInRtStatHide(ADR(tyP0938MagAW.tyMagAW3.tyBtnMtrGearEngage.uiMaskRtStat));
	END_IF

	//Interlock Limit Sensor
	IF tyP0938MagAW.tyMotionStd3.tyBtnOpenLmtSen.bValue = TRUE THEN
		fUIInRtStatOff(ADR(tyP0938MagAW.tyMotionStd3.tyBtnJogOpen.uiMaskRtStat));
	END_IF

	IF tyP0938MagAW.tyMotionStd3.tyBtnCloseLmtSen.bValue = TRUE THEN
		fUIInRtStatOff(ADR(tyP0938MagAW.tyMotionStd3.tyBtnJogClose.uiMaskRtStat));
	END_IF

	//Interlock When Moving
	IF tyP0938MagAW.tyMotionStd3.tyBtnOrigin.bRtCompl = TRUE THEN
		fUIInRtStatOff(ADR(tyP0938MagAW.tyMotionStd3.tyBtnMovAbs.uiMaskRtStat));
		fUIInRtStatOff(ADR(tyP0938MagAW.tyMotionStd3.tyBtnMovRel.uiMaskRtStat));
		fUIInRtStatOff(ADR(tyP0938MagAW.tyMotionStd3.tyBtnJogOpen.uiMaskRtStat));
		fUIInRtStatOff(ADR(tyP0938MagAW.tyMotionStd3.tyBtnJogClose.uiMaskRtStat));
		fUIInRtStatOff(ADR(tyP0938MagAW.tyMagAW3.tyBtnGo.uiMaskRtStat));
		fUIInRtStatOff(ADR(tyP0938MagAW.tyMagAW3.tyBtnMtrGearEngage.uiMaskRtStat));

	ELSIF tyP0938MagAW.tyMotionStd3.tyBtnMovAbs.bRtCompl = TRUE THEN
		fUIInRtStatOff(ADR(tyP0938MagAW.tyMotionStd3.tyBtnOrigin.uiMaskRtStat));
		fUIInRtStatOff(ADR(tyP0938MagAW.tyMotionStd3.tyBtnMovRel.uiMaskRtStat));
		fUIInRtStatOff(ADR(tyP0938MagAW.tyMotionStd3.tyBtnJogOpen.uiMaskRtStat));
		fUIInRtStatOff(ADR(tyP0938MagAW.tyMotionStd3.tyBtnJogClose.uiMaskRtStat));
		fUIInRtStatOff(ADR(tyP0938MagAW.tyMagAW3.tyBtnGo.uiMaskRtStat));
		fUIInRtStatOff(ADR(tyP0938MagAW.tyMagAW3.tyBtnMtrGearEngage.uiMaskRtStat));

	ELSIF tyP0938MagAW.tyMotionStd3.tyBtnMovRel.bRtCompl = TRUE THEN
		fUIInRtStatOff(ADR(tyP0938MagAW.tyMotionStd3.tyBtnOrigin.uiMaskRtStat));
		fUIInRtStatOff(ADR(tyP0938MagAW.tyMotionStd3.tyBtnMovAbs.uiMaskRtStat));
		fUIInRtStatOff(ADR(tyP0938MagAW.tyMotionStd3.tyBtnJogOpen.uiMaskRtStat));
		fUIInRtStatOff(ADR(tyP0938MagAW.tyMotionStd3.tyBtnJogClose.uiMaskRtStat));
		fUIInRtStatOff(ADR(tyP0938MagAW.tyMagAW3.tyBtnGo.uiMaskRtStat));
		fUIInRtStatOff(ADR(tyP0938MagAW.tyMagAW3.tyBtnMtrGearEngage.uiMaskRtStat));

	ELSIF tyP0938MagAW.tyMotionStd3.tyBtnJogOpen.bRtCompl = TRUE OR tyP0938MagAW.tyMotionStd3.tyBtnJogOpen.bValue = TRUE THEN
		fUIInRtStatOff(ADR(tyP0938MagAW.tyMotionStd3.tyBtnOrigin.uiMaskRtStat));
		fUIInRtStatOff(ADR(tyP0938MagAW.tyMotionStd3.tyBtnMovAbs.uiMaskRtStat));
		fUIInRtStatOff(ADR(tyP0938MagAW.tyMotionStd3.tyBtnMovRel.uiMaskRtStat));
		fUIInRtStatOff(ADR(tyP0938MagAW.tyMotionStd3.tyBtnJogClose.uiMaskRtStat));
		fUIInRtStatOff(ADR(tyP0938MagAW.tyMagAW3.tyBtnGo.uiMaskRtStat));
		fUIInRtStatOff(ADR(tyP0938MagAW.tyMagAW3.tyBtnMtrGearEngage.uiMaskRtStat));

	ELSIF tyP0938MagAW.tyMotionStd3.tyBtnJogClose.bRtCompl = TRUE OR tyP0938MagAW.tyMotionStd3.tyBtnJogClose.bValue = TRUE THEN
		fUIInRtStatOff(ADR(tyP0938MagAW.tyMotionStd3.tyBtnOrigin.uiMaskRtStat));
		fUIInRtStatOff(ADR(tyP0938MagAW.tyMotionStd3.tyBtnMovAbs.uiMaskRtStat));
		fUIInRtStatOff(ADR(tyP0938MagAW.tyMotionStd3.tyBtnMovRel.uiMaskRtStat));
		fUIInRtStatOff(ADR(tyP0938MagAW.tyMotionStd3.tyBtnJogOpen.uiMaskRtStat));
		fUIInRtStatOff(ADR(tyP0938MagAW.tyMagAW3.tyBtnGo.uiMaskRtStat));
		fUIInRtStatOff(ADR(tyP0938MagAW.tyMagAW3.tyBtnMtrGearEngage.uiMaskRtStat));

	ELSIF tyP0938MagAW.tyMagAW3.tyBtnGo.bRtCompl = TRUE THEN
		fUIInRtStatOff(ADR(tyP0938MagAW.tyMotionStd3.tyBtnOrigin.uiMaskRtStat));
		fUIInRtStatOff(ADR(tyP0938MagAW.tyMotionStd3.tyBtnMovAbs.uiMaskRtStat));
		fUIInRtStatOff(ADR(tyP0938MagAW.tyMotionStd3.tyBtnMovRel.uiMaskRtStat));
		fUIInRtStatOff(ADR(tyP0938MagAW.tyMotionStd3.tyBtnJogOpen.uiMaskRtStat));
		fUIInRtStatOff(ADR(tyP0938MagAW.tyMotionStd3.tyBtnJogClose.uiMaskRtStat));
		fUIInRtStatOff(ADR(tyP0938MagAW.tyMagAW3.tyBtnMtrGearEngage.uiMaskRtStat));

	ELSIF tyP0938MagAW.tyMagAW3.tyBtnMtrGearEngage.bRtCompl = TRUE THEN
		fUIInRtStatOff(ADR(tyP0938MagAW.tyMotionStd3.tyBtnOrigin.uiMaskRtStat));
		fUIInRtStatOff(ADR(tyP0938MagAW.tyMotionStd3.tyBtnMovAbs.uiMaskRtStat));
		fUIInRtStatOff(ADR(tyP0938MagAW.tyMotionStd3.tyBtnMovRel.uiMaskRtStat));
		fUIInRtStatOff(ADR(tyP0938MagAW.tyMotionStd3.tyBtnJogOpen.uiMaskRtStat));
		fUIInRtStatOff(ADR(tyP0938MagAW.tyMotionStd3.tyBtnJogClose.uiMaskRtStat));
		fUIInRtStatOff(ADR(tyP0938MagAW.tyMagAW3.tyBtnGo.uiMaskRtStat));

	END_IF

	//Axis Error
	IF tyP0938MagAW.tyMotionStd3.tyBtnPwr.bRtCompl = TRUE THEN
		fUIInRtStatOff(ADR(tyP0938MagAW.tyMotionStd3.tyBtnRst.uiMaskRtStat));
	ELSE
		fUIInRtStatHide(ADR(tyP0938MagAW.tyMotionStd3.tyBtnRst.uiMaskRtStat));
	END_IF

	//Pneumatic
	IF tyP0938MagAW.tyMagAW3.tyBtnMtrGearEngage.bRtCompl = TRUE THEN
		fUIInRtStatOff(ADR(tyP0938MagAW.tyMagAW3.tyBtnEngage.uiMaskRtStat));
		fUIInRtStatOff(ADR(tyP0938MagAW.tyMagAW3.tyBtnDisengage.uiMaskRtStat));
	ELSE
		fUIInRtStatHide(ADR(tyP0938MagAW.tyMagAW3.tyBtnEngage.uiMaskRtStat));
		fUIInRtStatHide(ADR(tyP0938MagAW.tyMagAW3.tyBtnDisengage.uiMaskRtStat));
	END_IF

END_ACTION
```

#### Act_OptP0938UpdtDat.st
```iecst
ACTION Act_OptP0938UpdtDat:

	(*Magazine Auto Width 1*)
	tyP0938MagAW.tyMotionStd1.tyNumCurrPos.diValue			:= p_diMagAWOpen1ActualPos;
	tyP0938MagAW.tyMotionStd1.tyNumErrCode.diValue			:= UDINT_TO_DINT(p_udiMagAWOpen1AxisErrID);
	tyP0938MagAW.tyMotionStd1.tyBitmapPwr.usiValueIdx		:= BOOL_TO_USINT(p_bMagAWOpen1PwrOn);
	tyP0938MagAW.tyMotionStd1.tyBitmapRst.usiValueIdx		:= BOOL_TO_USINT(NOT p_bMagAWOpen1AxisErr);
	tyP0938MagAW.tyMotionStd1.tyBitmapOrigin.usiValueIdx	:= BOOL_TO_USINT(p_bMagAWOpen1IsHomed);
	tyP0938MagAW.tyMotionStd1.tyBtnOpenLmtSen.bValue		:= p_bMagAWOpen1OpenSen;
	tyP0938MagAW.tyMotionStd1.tyBtnCloseLmtSen.bValue		:= p_bMagAWOpen1CloseSen;

	tyP0938MagAW.tyMagAW1.tyBtnEngageRS.bValue		:= p_tyDI.bMag1WallEngageRS;
	tyP0938MagAW.tyMagAW1.tyBtnDisengageRS.bValue	:= p_tyDI.bMag1WallDisengageRS;

	//Machine Bitmap
	IF p_bMagAWOpen1IsHomed = TRUE THEN
		IF (p_diMagAWOpen1ActualPos + p_tyMcParamCurr.diMag1WidthAtHmPosInUM) <= (p_tyNtParamCurr.tyProdRcpWidth.diMax / 2) THEN
			tyP0938MagAW.tyMotionStd1.tyBitmapMc.uiValueIdx 	:= 283;
		ELSE
			tyP0938MagAW.tyMotionStd1.tyBitmapMc.uiValueIdx 	:= 281;
		END_IF
	ELSE
		tyP0938MagAW.tyMotionStd1.tyBitmapMc.uiValueIdx	:= 283;
	END_IF

	IF p_tyDI.bMag1WallEngageRS = TRUE THEN
		tyP0938MagAW.tyMotionStd1.tyBitmapMc.uiValueIdx	:= tyP0938MagAW.tyMotionStd1.tyBitmapMc.uiValueIdx + 1;
	END_IF

	IF p_tyNtParamCurr.eProjMag = ULMagDual THEN
		tyP0938MagAW.tyMotionStd1.tyBitmapMc.uiValueIdx	:= tyP0938MagAW.tyMotionStd1.tyBitmapMc.uiValueIdx + 100;
	END_IF

	(*Magazine Auto Width 2*)
	tyP0938MagAW.tyMotionStd2.tyNumCurrPos.diValue			:= p_diMagAWOpen2ActualPos;
	tyP0938MagAW.tyMotionStd2.tyNumErrCode.diValue			:= UDINT_TO_DINT(p_udiMagAWOpen2AxisErrID);
	tyP0938MagAW.tyMotionStd2.tyBitmapPwr.usiValueIdx		:= BOOL_TO_USINT(p_bMagAWOpen2PwrOn);
	tyP0938MagAW.tyMotionStd2.tyBitmapRst.usiValueIdx		:= BOOL_TO_USINT(NOT p_bMagAWOpen2AxisErr);
	tyP0938MagAW.tyMotionStd2.tyBitmapOrigin.usiValueIdx	:= BOOL_TO_USINT(p_bMagAWOpen2IsHomed);
	tyP0938MagAW.tyMotionStd2.tyBtnOpenLmtSen.bValue		:= p_bMagAWOpen2OpenSen;
	tyP0938MagAW.tyMotionStd2.tyBtnCloseLmtSen.bValue		:= p_bMagAWOpen2CloseSen;

	tyP0938MagAW.tyMagAW2.tyBtnEngageRS.bValue		:= p_tyDI.bMag2WallEngageRS;
	tyP0938MagAW.tyMagAW2.tyBtnDisengageRS.bValue	:= p_tyDI.bMag2WallDisengageRS;

	//Machine Bitmap
	IF p_bMagAWOpen2IsHomed = TRUE THEN
		IF (p_diMagAWOpen2ActualPos + p_tyMcParamCurr.diMag2WidthAtHmPosInUM) <= (p_tyNtParamCurr.tyProdRcpWidth.diMax / 2) THEN
			tyP0938MagAW.tyMotionStd2.tyBitmapMc.uiValueIdx 	:= 287;
		ELSE
			tyP0938MagAW.tyMotionStd2.tyBitmapMc.uiValueIdx 	:= 285;
		END_IF
	ELSE
		tyP0938MagAW.tyMotionStd2.tyBitmapMc.uiValueIdx	:= 287;
	END_IF

	IF p_tyDI.bMag2WallEngageRS = TRUE THEN
		tyP0938MagAW.tyMotionStd2.tyBitmapMc.uiValueIdx	:= tyP0938MagAW.tyMotionStd2.tyBitmapMc.uiValueIdx + 1;
	END_IF

	IF p_tyNtParamCurr.eProjMag = ULMagDual THEN
		tyP0938MagAW.tyMotionStd2.tyBitmapMc.uiValueIdx	:= tyP0938MagAW.tyMotionStd2.tyBitmapMc.uiValueIdx + 100;
	END_IF

	(*Magazine Auto Width 3*)
	tyP0938MagAW.tyMotionStd3.tyNumCurrPos.diValue			:= p_diMagAWOpen3ActualPos;
	tyP0938MagAW.tyMotionStd3.tyNumErrCode.diValue			:= UDINT_TO_DINT(p_udiMagAWOpen3AxisErrID);
	tyP0938MagAW.tyMotionStd3.tyBitmapPwr.usiValueIdx		:= BOOL_TO_USINT(p_bMagAWOpen3PwrOn);
	tyP0938MagAW.tyMotionStd3.tyBitmapRst.usiValueIdx		:= BOOL_TO_USINT(NOT p_bMagAWOpen3AxisErr);
	tyP0938MagAW.tyMotionStd3.tyBitmapOrigin.usiValueIdx	:= BOOL_TO_USINT(p_bMagAWOpen3IsHomed);
	tyP0938MagAW.tyMotionStd3.tyBtnOpenLmtSen.bValue		:= p_bMagAWOpen3OpenSen;
	tyP0938MagAW.tyMotionStd3.tyBtnCloseLmtSen.bValue		:= p_bMagAWOpen3CloseSen;

	tyP0938MagAW.tyMagAW3.tyBtnEngageRS.bValue		:= p_tyDI.bMag3WallEngageRS;
	tyP0938MagAW.tyMagAW3.tyBtnDisengageRS.bValue	:= p_tyDI.bMag3WallDisengageRS;

	//Machine Bitmap
	IF p_bMagAWOpen3IsHomed = TRUE THEN
		IF (p_diMagAWOpen3ActualPos + p_tyMcParamCurr.diMag3WidthAtHmPosInUM) <= (p_tyNtParamCurr.tyProdRcpWidth.diMax / 2) THEN
			tyP0938MagAW.tyMotionStd3.tyBitmapMc.uiValueIdx 	:= 291;
		ELSE
			tyP0938MagAW.tyMotionStd3.tyBitmapMc.uiValueIdx 	:= 289;
		END_IF
	ELSE
		tyP0938MagAW.tyMotionStd3.tyBitmapMc.uiValueIdx	:= 291;
	END_IF

	IF p_tyDI.bMag3WallEngageRS = TRUE THEN
		tyP0938MagAW.tyMotionStd3.tyBitmapMc.uiValueIdx	:= tyP0938MagAW.tyMotionStd3.tyBitmapMc.uiValueIdx + 1;
	END_IF

END_ACTION
```

#### Act_OptP0938Keypad.st
```iecst
ACTION Act_OptP0938Keypad:

	IF bDispMagAW1 = TRUE THEN

		(*Magazine Auto Width 1*)
		IF fUIOutRtStatTPIsOpen(ADR(tyP0938MagAW.tyMagAW1.tyNumNewWidth.uiRtStat)) = TRUE THEN
			tyProperty.tyKeypad.tyStringTitle.sKeypadTitle	:= tyP0938MagAW.tyMagAW1.tyNumNewWidth.sKeypadTitle;

		ELSIF fUIOutRtStatTPIsOpen(ADR(tyP0938MagAW.tyMotionStd1.tyNumTargetPos.uiRtStat)) = TRUE THEN
			tyProperty.tyKeypad.tyStringTitle.sKeypadTitle	:= tyP0938MagAW.tyMotionStd1.tyNumTargetPos.sKeypadTitle;

		ELSIF fUIOutRtStatTPIsOpen(ADR(tyP0938MagAW.tyMotionStd1.tyNumStepSize.uiRtStat)) = TRUE THEN
			tyProperty.tyKeypad.tyStringTitle.sKeypadTitle	:= tyP0938MagAW.tyMotionStd1.tyNumStepSize.sKeypadTitle;

		ELSIF fUIOutRtStatTPIsOpen(ADR(tyP0938MagAW.tyMotionStd1.tyNumNomSpd.uiRtStat)) = TRUE THEN
			tyProperty.tyKeypad.tyStringTitle.sKeypadTitle	:= tyP0938MagAW.tyMotionStd1.tyNumNomSpd.sKeypadTitle;

		ELSIF fUIOutRtStatTPIsOpen(ADR(tyP0938MagAW.tyMotionStd1.tyNumSlwSpd.uiRtStat)) = TRUE THEN
			tyProperty.tyKeypad.tyStringTitle.sKeypadTitle	:= tyP0938MagAW.tyMotionStd1.tyNumSlwSpd.sKeypadTitle;

		END_IF

	ELSIF bDispMagAW2 = TRUE THEN

		(*Magazine Auto Width 2*)
		IF fUIOutRtStatTPIsOpen(ADR(tyP0938MagAW.tyMagAW2.tyNumNewWidth.uiRtStat)) = TRUE THEN
			tyProperty.tyKeypad.tyStringTitle.sKeypadTitle	:= tyP0938MagAW.tyMagAW2.tyNumNewWidth.sKeypadTitle;

		ELSIF fUIOutRtStatTPIsOpen(ADR(tyP0938MagAW.tyMotionStd2.tyNumTargetPos.uiRtStat)) = TRUE THEN
			tyProperty.tyKeypad.tyStringTitle.sKeypadTitle	:= tyP0938MagAW.tyMotionStd2.tyNumTargetPos.sKeypadTitle;

		ELSIF fUIOutRtStatTPIsOpen(ADR(tyP0938MagAW.tyMotionStd2.tyNumStepSize.uiRtStat)) = TRUE THEN
			tyProperty.tyKeypad.tyStringTitle.sKeypadTitle	:= tyP0938MagAW.tyMotionStd2.tyNumStepSize.sKeypadTitle;

		ELSIF fUIOutRtStatTPIsOpen(ADR(tyP0938MagAW.tyMotionStd2.tyNumNomSpd.uiRtStat)) = TRUE THEN
			tyProperty.tyKeypad.tyStringTitle.sKeypadTitle	:= tyP0938MagAW.tyMotionStd2.tyNumNomSpd.sKeypadTitle;

		ELSIF fUIOutRtStatTPIsOpen(ADR(tyP0938MagAW.tyMotionStd2.tyNumSlwSpd.uiRtStat)) = TRUE THEN
			tyProperty.tyKeypad.tyStringTitle.sKeypadTitle	:= tyP0938MagAW.tyMotionStd2.tyNumSlwSpd.sKeypadTitle;

		END_IF

	ELSIF bDispMagAW3 = TRUE THEN

		(*Magazine Auto Width 3*)
		IF fUIOutRtStatTPIsOpen(ADR(tyP0938MagAW.tyMagAW3.tyNumNewWidth.uiRtStat)) = TRUE THEN
			tyProperty.tyKeypad.tyStringTitle.sKeypadTitle	:= tyP0938MagAW.tyMagAW3.tyNumNewWidth.sKeypadTitle;

		ELSIF fUIOutRtStatTPIsOpen(ADR(tyP0938MagAW.tyMotionStd3.tyNumTargetPos.uiRtStat)) = TRUE THEN
			tyProperty.tyKeypad.tyStringTitle.sKeypadTitle	:= tyP0938MagAW.tyMotionStd3.tyNumTargetPos.sKeypadTitle;

		ELSIF fUIOutRtStatTPIsOpen(ADR(tyP0938MagAW.tyMotionStd3.tyNumStepSize.uiRtStat)) = TRUE THEN
			tyProperty.tyKeypad.tyStringTitle.sKeypadTitle	:= tyP0938MagAW.tyMotionStd3.tyNumStepSize.sKeypadTitle;

		ELSIF fUIOutRtStatTPIsOpen(ADR(tyP0938MagAW.tyMotionStd3.tyNumNomSpd.uiRtStat)) = TRUE THEN
			tyProperty.tyKeypad.tyStringTitle.sKeypadTitle	:= tyP0938MagAW.tyMotionStd3.tyNumNomSpd.sKeypadTitle;

		ELSIF fUIOutRtStatTPIsOpen(ADR(tyP0938MagAW.tyMotionStd3.tyNumSlwSpd.uiRtStat)) = TRUE THEN
			tyProperty.tyKeypad.tyStringTitle.sKeypadTitle	:= tyP0938MagAW.tyMotionStd3.tyNumSlwSpd.sKeypadTitle;

		END_IF

	END_IF

	IF p_tyNtParamCurr.bMagAutoVerifyPrep THEN
		CASE p_tyMagRcpCurrRcp.usiMagModel OF
			0,1:
				tyP0938MagAW.tyMagAW1.tyNumNewWidth.diValueMax		:= p_tyNtParamCurr.tyProdRcpWidth.diMax-70000;
				tyP0938MagAW.tyMagAW2.tyNumNewWidth.diValueMax		:= p_tyNtParamCurr.tyProdRcpWidth.diMax-70000;
				tyP0938MagAW.tyMagAW3.tyNumNewWidth.diValueMax		:= p_tyNtParamCurr.tyProdRcpWidth.diMax-70000;

			2:
				tyP0938MagAW.tyMagAW1.tyNumNewWidth.diValueMax		:= p_tyNtParamCurr.tyProdRcpWidth.diMax;
				tyP0938MagAW.tyMagAW2.tyNumNewWidth.diValueMax		:= p_tyNtParamCurr.tyProdRcpWidth.diMax;
				tyP0938MagAW.tyMagAW3.tyNumNewWidth.diValueMax		:= p_tyNtParamCurr.tyProdRcpWidth.diMax;
		END_CASE
	ELSE
		tyP0938MagAW.tyMagAW1.tyNumNewWidth.diValueMax		:= p_tyNtParamCurr.tyProdRcpWidth.diMax;
		tyP0938MagAW.tyMagAW2.tyNumNewWidth.diValueMax		:= p_tyNtParamCurr.tyProdRcpWidth.diMax;
		tyP0938MagAW.tyMagAW3.tyNumNewWidth.diValueMax		:= p_tyNtParamCurr.tyProdRcpWidth.diMax;

	END_IF
END_ACTION
```

#### Act_OptP0938RstMnl.st
```iecst
ACTION Act_OptP0938RstMnl:

	(*Magazine Auto Width 1*)
	IF EDGEPOS((bManualMod = FALSE) OR (p_eMagAWOpen1Status = Error)) THEN

		eMagAWOpen1Act	:= MagAWActIdle;

		bJogSlow				:= FALSE;
		bJogFast				:= FALSE;
		fbJogSlowToFastDlyTm.IN	:= FALSE;

		tyP0938MagAW.tyMagAW1.tyBtnGo.bRtCompl					:= FALSE;
		tyP0938MagAW.tyMagAW1.tyBtnGo.bValue					:= FALSE;
		tyP0938MagAW.tyMagAW1.tyBtnGo.bRtLk						:= FALSE;
		tyP0938MagAW.tyMagAW1.tyBtnGo.uiMaskRtStat.0			:= FALSE;

		tyP0938MagAW.tyMagAW1.tyBtnMtrGearEngage.bRtCompl		:= FALSE;
		tyP0938MagAW.tyMagAW1.tyBtnMtrGearEngage.bValue			:= FALSE;
		tyP0938MagAW.tyMagAW1.tyBtnMtrGearEngage.bRtLk			:= FALSE;
		tyP0938MagAW.tyMagAW1.tyBtnMtrGearEngage.uiMaskRtStat.0	:= FALSE;

		tyP0938MagAW.tyMotionStd1.tyBtnPwr.bRtCompl				:= FALSE;
		tyP0938MagAW.tyMotionStd1.tyBtnStop.bRtCompl			:= FALSE;
		tyP0938MagAW.tyMotionStd1.tyBtnOrigin.bRtCompl			:= FALSE;
		tyP0938MagAW.tyMotionStd1.tyBtnRst.bRtCompl				:= FALSE;
		tyP0938MagAW.tyMotionStd1.tyBtnMovAbs.bRtCompl			:= FALSE;
		tyP0938MagAW.tyMotionStd1.tyBtnMovRel.bRtCompl			:= FALSE;
		tyP0938MagAW.tyMotionStd1.tyBtnJogOpen.bRtCompl			:= FALSE;
		tyP0938MagAW.tyMotionStd1.tyBtnJogClose.bRtCompl		:= FALSE;

		tyP0938MagAW.tyMotionStd1.tyBtnPwr.bValue				:= FALSE;
		tyP0938MagAW.tyMotionStd1.tyBtnStop.bValue				:= TRUE;
		tyP0938MagAW.tyMotionStd1.tyBtnOrigin.bValue			:= FALSE;
		tyP0938MagAW.tyMotionStd1.tyBtnRst.bValue				:= FALSE;
		tyP0938MagAW.tyMotionStd1.tyBtnMovAbs.bValue			:= FALSE;
		tyP0938MagAW.tyMotionStd1.tyBtnMovRel.bValue			:= FALSE;
		tyP0938MagAW.tyMotionStd1.tyBtnJogOpen.bValue			:= FALSE;
		tyP0938MagAW.tyMotionStd1.tyBtnJogClose.bValue			:= FALSE;

		tyP0938MagAW.tyMotionStd1.tyBtnPwr.bRtLk				:= FALSE;
		tyP0938MagAW.tyMotionStd1.tyBtnStop.bRtLk				:= TRUE;
		tyP0938MagAW.tyMotionStd1.tyBtnOrigin.bRtLk				:= FALSE;
		tyP0938MagAW.tyMotionStd1.tyBtnRst.bRtLk				:= FALSE;
		tyP0938MagAW.tyMotionStd1.tyBtnMovAbs.bRtLk				:= FALSE;
		tyP0938MagAW.tyMotionStd1.tyBtnMovRel.bRtLk				:= FALSE;
		tyP0938MagAW.tyMotionStd1.tyBtnJogOpen.bRtLk			:= FALSE;
		tyP0938MagAW.tyMotionStd1.tyBtnJogClose.bRtLk			:= FALSE;

		tyP0938MagAW.tyMotionStd1.tyBtnPwr.uiMaskRtStat			:= TRUE;
		tyP0938MagAW.tyMotionStd1.tyBtnOrigin.uiMaskRtStat		:= FALSE;
		tyP0938MagAW.tyMotionStd1.tyBtnRst.uiMaskRtStat			:= TRUE;
		tyP0938MagAW.tyMotionStd1.tyBtnMovAbs.uiMaskRtStat		:= FALSE;
		tyP0938MagAW.tyMotionStd1.tyBtnMovRel.uiMaskRtStat		:= FALSE;
		tyP0938MagAW.tyMotionStd1.tyBtnJogOpen.uiMaskRtStat		:= FALSE;
		tyP0938MagAW.tyMotionStd1.tyBtnJogClose.uiMaskRtStat	:= FALSE;

	END_IF

	IF EDGEPOS((bManualMod = FALSE) OR (p_eMag1AWEngageStatus = Error)) THEN

		eMag1AWEngageAct	:= PneuActIdle;

		tyP0938MagAW.tyMagAW1.tyBtnEngage.bRtCompl		:= FALSE;
		tyP0938MagAW.tyMagAW1.tyBtnEngage.bValue		:= FALSE;
		tyP0938MagAW.tyMagAW1.tyBtnDisengage.bRtCompl	:= FALSE;
		tyP0938MagAW.tyMagAW1.tyBtnDisengage.bValue		:= FALSE;

	END_IF

	(*Magazine Auto Width 2*)
	IF EDGEPOS((bManualMod = FALSE) OR (p_eMagAWOpen2Status = Error)) THEN

		eMagAWOpen2Act	:= MagAWActIdle;

		bJogSlow				:= FALSE;
		bJogFast				:= FALSE;
		fbJogSlowToFastDlyTm.IN	:= FALSE;

		tyP0938MagAW.tyMagAW2.tyBtnGo.bRtCompl					:= FALSE;
		tyP0938MagAW.tyMagAW2.tyBtnGo.bValue					:= FALSE;
		tyP0938MagAW.tyMagAW2.tyBtnGo.bRtLk						:= FALSE;
		tyP0938MagAW.tyMagAW2.tyBtnGo.uiMaskRtStat.0			:= FALSE;

		tyP0938MagAW.tyMagAW2.tyBtnMtrGearEngage.bRtCompl		:= FALSE;
		tyP0938MagAW.tyMagAW2.tyBtnMtrGearEngage.bValue			:= FALSE;
		tyP0938MagAW.tyMagAW2.tyBtnMtrGearEngage.bRtLk			:= FALSE;
		tyP0938MagAW.tyMagAW2.tyBtnMtrGearEngage.uiMaskRtStat.0	:= FALSE;

		tyP0938MagAW.tyMotionStd2.tyBtnPwr.bRtCompl				:= FALSE;
		tyP0938MagAW.tyMotionStd2.tyBtnStop.bRtCompl			:= FALSE;
		tyP0938MagAW.tyMotionStd2.tyBtnOrigin.bRtCompl			:= FALSE;
		tyP0938MagAW.tyMotionStd2.tyBtnRst.bRtCompl				:= FALSE;
		tyP0938MagAW.tyMotionStd2.tyBtnMovAbs.bRtCompl			:= FALSE;
		tyP0938MagAW.tyMotionStd2.tyBtnMovRel.bRtCompl			:= FALSE;
		tyP0938MagAW.tyMotionStd2.tyBtnJogOpen.bRtCompl			:= FALSE;
		tyP0938MagAW.tyMotionStd2.tyBtnJogClose.bRtCompl		:= FALSE;

		tyP0938MagAW.tyMotionStd2.tyBtnPwr.bValue				:= FALSE;
		tyP0938MagAW.tyMotionStd2.tyBtnStop.bValue				:= TRUE;
		tyP0938MagAW.tyMotionStd2.tyBtnOrigin.bValue			:= FALSE;
		tyP0938MagAW.tyMotionStd2.tyBtnRst.bValue				:= FALSE;
		tyP0938MagAW.tyMotionStd2.tyBtnMovAbs.bValue			:= FALSE;
		tyP0938MagAW.tyMotionStd2.tyBtnMovRel.bValue			:= FALSE;
		tyP0938MagAW.tyMotionStd2.tyBtnJogOpen.bValue			:= FALSE;
		tyP0938MagAW.tyMotionStd2.tyBtnJogClose.bValue			:= FALSE;

		tyP0938MagAW.tyMotionStd2.tyBtnPwr.bRtLk				:= FALSE;
		tyP0938MagAW.tyMotionStd2.tyBtnStop.bRtLk				:= TRUE;
		tyP0938MagAW.tyMotionStd2.tyBtnOrigin.bRtLk				:= FALSE;
		tyP0938MagAW.tyMotionStd2.tyBtnRst.bRtLk				:= FALSE;
		tyP0938MagAW.tyMotionStd2.tyBtnMovAbs.bRtLk				:= FALSE;
		tyP0938MagAW.tyMotionStd2.tyBtnMovRel.bRtLk				:= FALSE;
		tyP0938MagAW.tyMotionStd2.tyBtnJogOpen.bRtLk			:= FALSE;
		tyP0938MagAW.tyMotionStd2.tyBtnJogClose.bRtLk			:= FALSE;

		tyP0938MagAW.tyMotionStd2.tyBtnPwr.uiMaskRtStat			:= TRUE;
		tyP0938MagAW.tyMotionStd2.tyBtnOrigin.uiMaskRtStat		:= FALSE;
		tyP0938MagAW.tyMotionStd2.tyBtnRst.uiMaskRtStat			:= TRUE;
		tyP0938MagAW.tyMotionStd2.tyBtnMovAbs.uiMaskRtStat		:= FALSE;
		tyP0938MagAW.tyMotionStd2.tyBtnMovRel.uiMaskRtStat		:= FALSE;
		tyP0938MagAW.tyMotionStd2.tyBtnJogOpen.uiMaskRtStat		:= FALSE;
		tyP0938MagAW.tyMotionStd2.tyBtnJogClose.uiMaskRtStat	:= FALSE;

	END_IF

	IF EDGEPOS((bManualMod = FALSE) OR (p_eMag2AWEngageStatus = Error)) THEN

		eMag2AWEngageAct	:= PneuActIdle;

		tyP0938MagAW.tyMagAW2.tyBtnEngage.bRtCompl		:= FALSE;
		tyP0938MagAW.tyMagAW2.tyBtnEngage.bValue		:= FALSE;
		tyP0938MagAW.tyMagAW2.tyBtnDisengage.bRtCompl	:= FALSE;
		tyP0938MagAW.tyMagAW2.tyBtnDisengage.bValue		:= FALSE;

	END_IF

	(*Magazine Auto Width 3*)
	IF EDGEPOS((bManualMod = FALSE) OR (p_eMagAWOpen3Status = Error)) THEN

		eMagAWOpen3Act	:= MagAWActIdle;

		bJogSlow				:= FALSE;
		bJogFast				:= FALSE;
		fbJogSlowToFastDlyTm.IN	:= FALSE;

		tyP0938MagAW.tyMagAW3.tyBtnGo.bRtCompl					:= FALSE;
		tyP0938MagAW.tyMagAW3.tyBtnGo.bValue					:= FALSE;
		tyP0938MagAW.tyMagAW3.tyBtnGo.bRtLk						:= FALSE;
		tyP0938MagAW.tyMagAW3.tyBtnGo.uiMaskRtStat.0			:= FALSE;

		tyP0938MagAW.tyMagAW3.tyBtnMtrGearEngage.bRtCompl		:= FALSE;
		tyP0938MagAW.tyMagAW3.tyBtnMtrGearEngage.bValue			:= FALSE;
		tyP0938MagAW.tyMagAW3.tyBtnMtrGearEngage.bRtLk			:= FALSE;
		tyP0938MagAW.tyMagAW3.tyBtnMtrGearEngage.uiMaskRtStat.0	:= FALSE;

		tyP0938MagAW.tyMotionStd3.tyBtnPwr.bRtCompl				:= FALSE;
		tyP0938MagAW.tyMotionStd3.tyBtnStop.bRtCompl			:= FALSE;
		tyP0938MagAW.tyMotionStd3.tyBtnOrigin.bRtCompl			:= FALSE;
		tyP0938MagAW.tyMotionStd3.tyBtnRst.bRtCompl				:= FALSE;
		tyP0938MagAW.tyMotionStd3.tyBtnMovAbs.bRtCompl			:= FALSE;
		tyP0938MagAW.tyMotionStd3.tyBtnMovRel.bRtCompl			:= FALSE;
		tyP0938MagAW.tyMotionStd3.tyBtnJogOpen.bRtCompl			:= FALSE;
		tyP0938MagAW.tyMotionStd3.tyBtnJogClose.bRtCompl		:= FALSE;

		tyP0938MagAW.tyMotionStd3.tyBtnPwr.bValue				:= FALSE;
		tyP0938MagAW.tyMotionStd3.tyBtnStop.bValue				:= TRUE;
		tyP0938MagAW.tyMotionStd3.tyBtnOrigin.bValue			:= FALSE;
		tyP0938MagAW.tyMotionStd3.tyBtnRst.bValue				:= FALSE;
		tyP0938MagAW.tyMotionStd3.tyBtnMovAbs.bValue			:= FALSE;
		tyP0938MagAW.tyMotionStd3.tyBtnMovRel.bValue			:= FALSE;
		tyP0938MagAW.tyMotionStd3.tyBtnJogOpen.bValue			:= FALSE;
		tyP0938MagAW.tyMotionStd3.tyBtnJogClose.bValue			:= FALSE;

		tyP0938MagAW.tyMotionStd3.tyBtnPwr.bRtLk				:= FALSE;
		tyP0938MagAW.tyMotionStd3.tyBtnStop.bRtLk				:= TRUE;
		tyP0938MagAW.tyMotionStd3.tyBtnOrigin.bRtLk				:= FALSE;
		tyP0938MagAW.tyMotionStd3.tyBtnRst.bRtLk				:= FALSE;
		tyP0938MagAW.tyMotionStd3.tyBtnMovAbs.bRtLk				:= FALSE;
		tyP0938MagAW.tyMotionStd3.tyBtnMovRel.bRtLk				:= FALSE;
		tyP0938MagAW.tyMotionStd3.tyBtnJogOpen.bRtLk			:= FALSE;
		tyP0938MagAW.tyMotionStd3.tyBtnJogClose.bRtLk			:= FALSE;

		tyP0938MagAW.tyMotionStd3.tyBtnPwr.uiMaskRtStat			:= TRUE;
		tyP0938MagAW.tyMotionStd3.tyBtnOrigin.uiMaskRtStat		:= FALSE;
		tyP0938MagAW.tyMotionStd3.tyBtnRst.uiMaskRtStat			:= TRUE;
		tyP0938MagAW.tyMotionStd3.tyBtnMovAbs.uiMaskRtStat		:= FALSE;
		tyP0938MagAW.tyMotionStd3.tyBtnMovRel.uiMaskRtStat		:= FALSE;
		tyP0938MagAW.tyMotionStd3.tyBtnJogOpen.uiMaskRtStat		:= FALSE;
		tyP0938MagAW.tyMotionStd3.tyBtnJogClose.uiMaskRtStat	:= FALSE;

	END_IF

	IF EDGEPOS((bManualMod = FALSE) OR (p_eMag3AWEngageStatus = Error)) THEN

		eMag3AWEngageAct	:= PneuActIdle;

		tyP0938MagAW.tyMagAW3.tyBtnEngage.bRtCompl		:= FALSE;
		tyP0938MagAW.tyMagAW3.tyBtnEngage.bValue		:= FALSE;
		tyP0938MagAW.tyMagAW3.tyBtnDisengage.bRtCompl	:= FALSE;
		tyP0938MagAW.tyMagAW3.tyBtnDisengage.bValue		:= FALSE;

	END_IF

END_ACTION
```

#### Act_EntP0939Disp.st
```iecst
ACTION Act_EntP0939Disp:

	//Access Address
	p_tyC0001MotionStd ACCESS ADR(tyP0939Lifter2.tyMotionStd);

	p_tyC0002FullMask ACCESS ADR(tyP0939Lifter2.tyFullMaskHide);

	p_tyC0004Navi ACCESS ADR(tyP0939Lifter2.tyNaviBack);

	p_tyC0005Main ACCESS ADR(tyCommon.tyMain);

	p_tyC0007Notif ACCESS ADR(tyCommon.tyNotif);

	p_tyC0008MsgBox ACCESS ADR(tyP0939Lifter2.tyMsgBoxHide);

	p_tyC0009Info ACCESS ADR(tyCommon.tyInfo);

	p_tyP0939Lifter ACCESS ADR(tyP0939Lifter2.tyLifter);

//	p_tyP0939InOutletShutterFB ACCESS ADR(tyP0939Lifter2.tyInOutletShutterFB);

	//Display
	tyP0939Lifter2.tyMotionStd.tyBtnPwr.bValue	:= p_bLifter2PwrOn;

	tyP0939Lifter2.tyLifter.tyNumNewSlt.diValueMax	:= p_tyMagRcpCurrRcp.diTtlSlt;

END_ACTION
```

#### Act_OptP0939Navi.st
```iecst
ACTION Act_OptP0939Navi:

	IF tyP0939Lifter2.tyNaviBack.tyBtnBack.bRtCompl = TRUE THEN
		tyP0939Lifter2.tyNaviBack.tyBtnBack.bRtCompl	:= FALSE;
		tyP0939Lifter2.tyNaviBack.tyBtnBack.bValue	:= FALSE;

		eChgPage	:= UIP0920MtrNPneuCtrl;

	END_IF

END_ACTION
```

#### Act_OptP0939FullMask.st
```iecst
ACTION Act_OptP0939FullMask:

	IF eCurrPage = UIP0939Lifter2 THEN

		IF p_tyDI.bEStopSig = FALSE THEN
			p_tyC0002FullMask ACCESS ADR(tyP0939Lifter2.tyFullMaskEStop);

		ELSIF p_tyDI.bCoverSWSig = FALSE THEN
			p_tyC0002FullMask ACCESS ADR(tyP0939Lifter2.tyFullMaskCWSig);

		ELSIF p_tyDI.bSafetyRlySig = FALSE THEN
			p_tyC0002FullMask ACCESS ADR(tyP0939Lifter2.tyFullMaskSafetyRly);

		ELSIF p_tyDI.bPusherExtRS = TRUE THEN
			p_tyC0002FullMask ACCESS ADR(tyP0939Lifter2.tyFullMaskPshrInterrupt);

//		ELSIF p_tyNtParamCurr.bProjInletShutPrep AND p_tyDI.bInShutterCloseRS = FALSE THEN
//			p_tyC0002FullMask ACCESS ADR(tyP0939Lifter2.tyFullMaskInShutOpnInterrupt);

		ELSIF p_tyNtParamCurr.bProjOutletShutPrep AND p_tyDI.bOutShutterCloseRS = FALSE THEN
			p_tyC0002FullMask ACCESS ADR(tyP0939Lifter2.tyFullMaskOutShutOpnInterrupt);

		ELSIF p_tyDI.bConvLftSen THEN
			p_tyC0002FullMask ACCESS ADR(tyP0939Lifter2.tyFullMaskLftSenInterrupt);

		ELSIF p_tyDI.bConvClrSen THEN
			p_tyC0002FullMask ACCESS ADR(tyP0939Lifter2.tyFullMaskClrSenInterrupt);

		ELSIF p_tyDI.bLifterSafetyLmtSW1 = FALSE OR p_tyDI.bLifterSafetyLmtSW2 = FALSE THEN
			p_tyC0002FullMask ACCESS ADR(tyP0939Lifter2.tyFullMaskSafetyLmtSW);

		ELSIF p_tyDI.bLifterTimingBeltSen = FALSE THEN
			p_tyC0002FullMask ACCESS ADR(tyP0939Lifter2.tyFullMaskTimingBelt);

		ELSIF p_tyNtParamCurr.tyDISettings.diMag2FixedClampRS <> 0 AND p_tyDI.bMag2FixedClampRS = FALSE
			AND p_tyDI.bMagPresentSen1 THEN
			p_tyC0002FullMask ACCESS ADR(tyP0939Lifter2.tyFullMaskMagClmpInt);

		ELSE
			p_tyC0002FullMask ACCESS ADR(tyP0939Lifter2.tyFullMaskHide);

		END_IF

	END_IF

END_ACTION
```
